{attribute 'ac_persist' := 'PersistenceChannel'}
Low_temperature_alarm_differential : REAL ;
{attribute 'ac_persist' := 'PersistenceChannel'}
High_temperature_alarm_differential : REAL ;
{attribute 'ac_persist' := 'PersistenceChannel'}
Probe_used_for_temperature_alarm_detection : REAL ;
{attribute 'ac_persist' := 'PersistenceChannel'}
Temperature_alarm_delay : REAL ;
Temperature_alarm_delay_write_int : INT ;
{attribute 'ac_persist' := 'PersistenceChannel'}
Operation_in_case_of_high_condenser_alarm : REAL ;
{attribute 'ac_persist' := 'PersistenceChannel'}
Condensation_temperature_alarm : REAL ;
{attribute 'ac_persist' := 'PersistenceChannel'}
Standby_button_enabling : REAL ;
{attribute 'ac_persist' := 'PersistenceChannel'}
Door_switch_input_mode : REAL ;
Door_switch_input_mode_write_int : INT ;
{attribute 'ac_persist' := 'PersistenceChannel'}
Door_alarm_delay : REAL ;
Door_alarm_delay_write_int : INT ;
{attribute 'ac_persist' := 'PersistenceChannel'}
Compressor_stop_delay : REAL ;
Compressor_stop_delay_write_int : INT ;
{attribute 'ac_persist' := 'PersistenceChannel'}
Door_stop_timeout : REAL ;
Door_stop_timeout_write_int : INT ;
{attribute 'ac_persist' := 'PersistenceChannel'}
DI1_digital_input_operation : REAL ;
{attribute 'ac_persist' := 'PersistenceChannel'}
DI1_digital_input_activation : REAL ;
{attribute 'ac_persist' := 'PersistenceChannel'}
DI2_digital_input_operation : REAL ;
{attribute 'ac_persist' := 'PersistenceChannel'}
DI2_digital_input_activation : REAL ;
DI1_digital_input_operation_write_int : INT ;
DI1_digital_input_activation_write_int : INT ;
DI2_digital_input_operation_write_int : INT ;
DI2_digital_input_activation_write_int : INT ;
{attribute 'ac_persist' := 'PersistenceChannel'}
Light_control_mode : REAL ;
Light_control_mode_write_int : INT ;
{attribute 'ac_persist' := 'PersistenceChannel'}
standby : REAL;
standby_write : INT;
{attribute 'ac_persist' := 'PersistenceChannel'}
Light_control : REAL;

write_data_alarm : R_TRIG;
write_data_setp : R_TRIG;
write_data_defrost : R_TRIG;
write_data_mute : R_TRIG;
write_data_control : R_TRIG;
write_data_man_defrost : R_TRIG;
door_open_trigger : R_TRIG ;
door_close_trigger : F_TRIG ;
set_param_trigger : R_TRIG ;
get_param_trigger : R_TRIG ;
all_param_read : BOOL ;
no_loop : INT :=0 ;


control_button : BOOL  := TRUE ;
defrost_button : BOOL  := FALSE ;
setpoint_button : BOOL ;
read_param_button : BOOL ;
{attribute 'ac_persist' := 'PersistenceChannel'}
RL1_output_operation : REAL ;
{attribute 'ac_persist' := 'PersistenceChannel'}
RL2_output_operation : REAL ;
{attribute 'ac_persist' := 'PersistenceChannel'}
RL3_output_operation : REAL ;
{attribute 'ac_persist' := 'PersistenceChannel'}
RL4_output_operation : REAL ;
RL1_output_operation_write_int : INT ;
RL2_output_operation_write_int : INT ;
RL3_output_operation_write_int : INT ;
RL4_output_operation_write_int : INT ;
{attribute 'ac_persist' := 'PersistenceChannel'}
Probe_T1_offset : REAL ;
{attribute 'ac_persist' := 'PersistenceChannel'}
Probe_T2_enable : REAL ;
{attribute 'ac_persist' := 'PersistenceChannel'}
Probe_T2_offset : REAL ;
{attribute 'ac_persist' := 'PersistenceChannel'}
Auxiliary_probe_T3_operation : REAL ;
{attribute 'ac_persist' := 'PersistenceChannel'}
Probe_T3_offset : REAL ;
{attribute 'ac_persist' := 'PersistenceChannel'}
Delay_for_minimum_and_maximum_temperature_logging : REAL ;
{attribute 'ac_persist' := 'PersistenceChannel'}
Selects_the_temperature_probe_to_be_displayed : REAL ;
{attribute 'ac_persist' := 'PersistenceChannel'}
The_relative_weight_of_T2_on_T1 : REAL ;
{attribute 'ac_persist' := 'PersistenceChannel'}
Display_slowdown : REAL ;
Display_slowdown_write_int : INT ;
{attribute 'ac_persist' := 'PersistenceChannel'}
Address_for_PC_communication : REAL ;
Address_for_PC_communication_write_int : INT ;
{attribute 'ac_persist' := 'PersistenceChannel'}
Modbus_protocol_selection : REAL ;
Modbus_protocol_selection_write_int : INT ;
// Word variables
Status_BITs_0_to_15 : WORD;
Status_BITs_16_to_31 : WORD;
Alarm_BITs_0_to_15 : WORD;
setp_write_word : WORD ;
Fan_stop_temperature_write_word : WORD ;

dig1 : BOOL;
dig2 : BOOL;
dout1 : BOOL;
dout2 : BOOL;
dout3 : BOOL;
dout4 : BOOL;
alarm : BOOL;
buzzer_mute : BOOL;
defrost : BOOL;
door_open : BOOL;
test : BOOL;
machine_standby : BOOL;
T1_failure  : BOOL;
T2_failure  : BOOL;
T3_failure  : BOOL;
Low_temperature  : BOOL;
High_temperature  : BOOL;
High_condenser_temperature  : BOOL;
Generic_alarm  : BOOL;
Door_open_alarm  : BOOL;
RL1 : BOOL;
RL2 : BOOL;
RL3 : BOOL;
SSR : BOOL;
deactivate_defrost_button : BOOL ;
modbus_communication : BOOL ;
comm_indicator : REAL ;



//triggers for writing setpoints and parameters
xtrigger_alarm : BOOL;
xtrigger_setp : BOOL;
xtrigger_defrost : BOOL;
xtrigger_mute : BOOL;
xtrigger_control : BOOL;
xtrigger_man_defrost : BOOL;
xtrigger_get_param : BOOL;
xtrigger_set_param : BOOL;







//Graphic variables
Unit_switch_status : INT;
i : INT;
show_trendvalue : ARRAY[0..50] OF BOOL;
select_trendvalue : INT :=0 ;

END_VAR




temp_provision_room:= scaleFunction(modbus_var[0],0.1, 0);
temp_defrost := scaleFunction(modbus_var[1],0.1, 0);
reg2 := scaleFunction(modbus_var[2],0.1, 0); // not used ?
reg3 := scaleFunction(modbus_var[3],0.1, 0); // not used ?
reg4 := scaleFunction(modbus_var[4],0.1, 0); // not used ?
reg5 := scaleFunction(modbus_var[5],0.1, 0); // not used ?
reg6 := scaleFunction(modbus_var[6],0.1, 0); // not used ?
reg7 := scaleFunction(modbus_var[7],0.1, 0); // not used ?
reg8 := scaleFunction(modbus_var[8],0.1, 0); // not used ?
reg9 := scaleFunction(modbus_var[9],0.1, 0); // not used ?
reg10 := modbus_var[10]; // not used ?
set_point := scaleFunction(modbus_var[11],0.1, 0);  // not used ?
reg12 := scaleFunction(modbus_var[12],0.1, 0); // not used ?
reg13 := scaleFunction(modbus_var[13],0.1, 0); // not used ?
reg14 := scaleFunction(modbus_var[14],0.1, 0); // not used ?
reg15 := scaleFunction(modbus_var[15],0.1, 0); // not used ?
reg16 := scaleFunction(modbus_var[16],0.1, 0); // not used ?
reg17 := scaleFunction(modbus_var[17],0.1, 0); // not used ?

// Non changeable parameters

T1_offset := scaleFunction(modbus_var1[2000],1, 0);
T2_offset := scaleFunction(modbus_var1[2001],1, 2);
T3_offset := scaleFunction(modbus_var1[2002],1, 3);
T1_span := scaleFunction(modbus_var1[2003],1, 4);
T2_span := scaleFunction(modbus_var1[2004],1, 5);
T3_span := scaleFunction(modbus_var1[2005],1, 6);

valore_tasto1_V := scaleFunction(modbus_var[150],1, 6);
valore_tasto_UP := scaleFunction(modbus_var[151],1, 6);
valore_tasto_DW := scaleFunction(modbus_var[152],1, 6);
valore_tasto_X := scaleFunction(modbus_var[153],1, 6);

Test_display := scaleFunction(modbus_var[193],1, 0);
Tasto_attualmente_premuto := scaleFunction(modbus_var[194],1, 0);
Password := scaleFunction(modbus_var[197],1, 0);

preset_parameters:= scaleFunction(modbus_var[200],1, 0);

Setpoint:= scaleFunction(modbus_var[303],0.1, 0);
Thermostat_OFF_ON_ref_to_SP:= scaleFunction(modbus_var[304],0.1, 0);
Thermostat_ON_OFF_ref_to_SP:= scaleFunction(modbus_var[305],0.1, 0);

Defrost_start_mode:= scaleFunction(modbus_var[400],1, 0);
Time_based_defrost:= scaleFunction(modbus_var[401],1, 0);

Delay_for_pressure_equalization_for_hot_gas:= scaleFunction(modbus_var[405],1, 0);

Defrost_end_temperature:= scaleFunction(modbus_var[406],0.1, 0);
Maximum_defrost_duration:= scaleFunction(modbus_var[407],1, 0);

Drain_down_time:= scaleFunction(modbus_var[408],1, 0);
Display_defrost_mode:= scaleFunction(modbus_var[409],1, 0);

Target_evaporator_temperature:= scaleFunction(modbus_var[453],0.1, 0);
Fan_stop_delay_after_compressor_stop:= scaleFunction(modbus_var[454],1, 0);
Timed_fan_stop:= scaleFunction(modbus_var[455],1, 0);
Timed_fan_run:= scaleFunction(modbus_var[456],1, 0);
Fan_Minimum_Stop:= scaleFunction(modbus_var[457],1, 0);


Low_temperature_alarm_threshold:= scaleFunction(modbus_var[501],0.1, 0);
High_temperature_alarm_threshold:= scaleFunction(modbus_var[502],0.1, 0);
Low_temperature_alarm_differential:= scaleFunction(modbus_var[503],0.1, 0);
High_temperature_alarm_differential:= scaleFunction(modbus_var[504],0.1, 0);
Probe_used_for_temperature_alarm_detection:= scaleFunction(modbus_var[505],1, 0);
Operation_in_case_of_high_condenser_alarm:= scaleFunction(modbus_var[507],1, 0);
Condensation_temperature_alarm:= scaleFunction(modbus_var[508],0.1, 0);

Standby_button_enabling:= scaleFunction(modbus_var[600],1, 0);



// Changeable parameters
delay_timer(IN:=read_param_button, PT:=set_delaytime);
IF read_param_button THEN
	Display_slowdown:= scaleFunction(modbus_var[208],1, 0);
	Readout_scale:= scaleFunction(modbus_var[300],1, 0);
	Minimum_temperature_setpoint:= scaleFunction(modbus_var[301],0.1, 0);
	Maximum_temperature_setpoint:= scaleFunction(modbus_var[302],0.1, 0);
	CH_minimum_OFF_time:= scaleFunction(modbus_var[306],1, 0);
	CH_minimum_ON_time:= scaleFunction(modbus_var[307],1, 0);
	CH_output_ON_when_probe_T1_is_faulty:= scaleFunction(modbus_var[308],1, 0);
	CH_output_OFF_when_probe_T1_is_faulty:= scaleFunction(modbus_var[309],1, 0);
	Minimum_Time_Between_Defrost:= scaleFunction(modbus_var[402],1, 0);
	Defrost_time_optimization:= scaleFunction(modbus_var[403],1, 0);
	Defrost_type:= scaleFunction(modbus_var[404],1, 0);
//	Defrost_end_temperature:= scaleFunction(modbus_var[406],1, 0);
//	Maximum_defrost_duration:= scaleFunction(modbus_var[407],1, 0);
	Display_delay:= scaleFunction(modbus_var[410],1, 0);
	Fans_active_during_defrost:= scaleFunction(modbus_var[411],1, 0);
	Fan_restart_temperature_after_defrost:= scaleFunction(modbus_var[412],0.1, 0);
	Fan_mode_during_thermostatic_control:= scaleFunction(modbus_var[452],1, 0);
	Fan_stop_temperature:= scaleFunction(modbus_var[450],0.1, 0);
	Maximum_fan_stop_for_FDD_FET:= scaleFunction(modbus_var[451],1, 0);
	Alarm_threshold_management:= scaleFunction(modbus_var[500],1, 0);
	Temperature_alarm_delay:= scaleFunction(modbus_var[506],1, 0);
	Door_switch_input_mode:= scaleFunction(modbus_var[601],1, 0);
	Door_alarm_delay:= scaleFunction(modbus_var[602],1, 0);
	Compressor_stop_delay:= scaleFunction(modbus_var[603],1, 0);
	Door_stop_timeout:= scaleFunction(modbus_var[604],1, 0);
	DI1_digital_input_operation:= scaleFunction(modbus_var[605],1, 0);
	DI1_digital_input_activation:= scaleFunction(modbus_var[606],1, 0);
	DI2_digital_input_operation:= scaleFunction(modbus_var[607],1, 0);
	DI2_digital_input_activation:= scaleFunction(modbus_var[608],1, 0);
	Light_control_mode:= scaleFunction(modbus_var[609],1, 0);
	RL1_output_operation:= scaleFunction(modbus_var[650],1, 0);
	RL2_output_operation:= scaleFunction(modbus_var[651],1, 0);
	RL3_output_operation:= scaleFunction(modbus_var[652],1, 0);
	RL4_output_operation:= scaleFunction(modbus_var[653],1, 0);

	// no_loop :=no_loop +1 ;
	IF delay_timer.Q THEN
		read_param_button := FALSE ;
		no_loop:=0;
	END_IF	
END_IF










standby:= scaleFunction(modbus_var[702],1, 0);
Light_control:= scaleFunction(modbus_var[703],1, 0);




Probe_T1_offset:= scaleFunction(modbus_var[201],0.1, 0);
Probe_T2_enable:= scaleFunction(modbus_var[202],1, 0);
Probe_T2_offset:= scaleFunction(modbus_var[203],0.1, 0);
Auxiliary_probe_T3_operation:= scaleFunction(modbus_var[204],1, 0);
Probe_T3_offset:= scaleFunction(modbus_var[205],0.1, 0);
Selects_the_temperature_probe_to_be_displayed:= scaleFunction(modbus_var[206],1, 0);
The_relative_weight_of_T2_on_T1:= scaleFunction(modbus_var[207],1, 0);

Address_for_PC_communication:= scaleFunction(modbus_var[209],1, 0);
Modbus_protocol_selection:= scaleFunction(modbus_var[210],1, 0);
Delay_for_minimum_and_maximum_temperature_logging:= scaleFunction(modbus_var[211],1, 0);

//  Statusbits
Status_BITs_0_to_15 := modbus_var[100];
Status_BITs_16_to_31 := modbus_var[102];
Alarm_BITs_0_to_15 := modbus_var[101];


alarm := maskbitFunction(Status_BITs_0_to_15,0) OR NOT modbus_communication ;
buzzer_mute := maskbitFunction(Status_BITs_0_to_15,1);
defrost:= maskbitFunction(Status_BITs_0_to_15,2);
door_open := maskbitFunction(Status_BITs_0_to_15,3);
test := maskbitFunction(Status_BITs_0_to_15,4);
machine_standby := maskbitFunction(Status_BITs_0_to_15,5);


T1_failure := maskbitFunction(Alarm_BITs_0_to_15,0);
T2_failure := maskbitFunction(Alarm_BITs_0_to_15,1);
T3_failure := maskbitFunction(Alarm_BITs_0_to_15,2);
Low_temperature := maskbitFunction(Alarm_BITs_0_to_15,3);
High_temperature := maskbitFunction(Alarm_BITs_0_to_15,4);
High_condenser_temperature := maskbitFunction(Alarm_BITs_0_to_15,5);
Generic_alarm := maskbitFunction(Alarm_BITs_0_to_15,6);
Door_open_alarm := maskbitFunction(Alarm_BITs_0_to_15,7);

dout1 := maskbitFunction(Status_BITs_16_to_31,0); 
dout2 := maskbitFunction(Status_BITs_16_to_31,1);
dout3 := maskbitFunction(Status_BITs_16_to_31,2);
dout4 := maskbitFunction(Status_BITs_16_to_31,3);

RL1 := maskbitFunction(modbus_var[196],0);
RL2 := maskbitFunction(modbus_var[196],1);

RL3 := maskbitFunction(modbus_var[196],2);
SSR := maskbitFunction(modbus_var[196],3);


dig1 := maskbitFunction(reg10,0);
dig2 := maskbitFunction(reg10,1);

// Communication fault
comm_indicator := temp_provision_room + temp_defrost + reg2 + reg3 + reg4 + reg5
+ reg6 + reg7 + reg8 + reg9 + reg10 ;
IF comm_indicator = 0 THEN
	modbus_communication := FALSE ;
ELSE
	modbus_communication := TRUE ;
END_IF
	



// Parameter write values

setp_write_word := REAL_TO_INT(setp_write*10) ;
Thermostat_OFF_ON_write_word := REAL_TO_INT(Thermostat_OFF_ON_write*10) ;
Thermostat_ON_OFF_write_word:= REAL_TO_INT(Thermostat_ON_OFF_write*10) ;
Low_temperature_alarm_thres_write_word:= REAL_TO_INT(Low_temperature_alarm_thres_write*10);
High_temperature_alarm_thres_write_word:= REAL_TO_INT(High_temperature_alarm_thres_write*10);
muteAlarm :=1 ;
Time_based_defrost_write_word:= REAL_TO_INT(Time_based_defrost_write*1);
Defrost_end_temperature_write_word:= REAL_TO_INT(Defrost_end_temperature_write*10);
Drain_down_time_write_int:= REAL_TO_INT(Drain_down_time_write);
Maximum_defrost_duration_write_word:= REAL_TO_INT(Maximum_defrost_duration_write*1);
Fan_stop_temperature_write_word:= REAL_TO_INT(Fan_stop_temperature*10);
preset_parameters_write_int:=REAL_TO_INT(preset_parameters);
Readout_scale_write_int:=REAL_TO_INT(Readout_scale);
Minimum_temperature_setpoint_write_int:=REAL_TO_INT(Minimum_temperature_setpoint*10);
Maximum_temperature_setpoint_write_int:=REAL_TO_INT(Maximum_temperature_setpoint*10);
CH_minimum_OFF_time_write_int:=REAL_TO_INT(CH_minimum_OFF_time);
CH_minimum_ON_time_write_int:=REAL_TO_INT(CH_minimum_ON_time);
CH_output_ON_when_probe_T1_is_faulty_write_int:=REAL_TO_INT(CH_output_ON_when_probe_T1_is_faulty);
CH_output_OFF_when_probe_T1_is_faulty_write_int:=REAL_TO_INT(CH_output_OFF_when_probe_T1_is_faulty);
Minimum_Time_Between_Defrost_write_int:=REAL_TO_INT(Minimum_Time_Between_Defrost);
Defrost_time_optimization_write_int:=REAL_TO_INT(Defrost_time_optimization);
Defrost_type_write_int:=REAL_TO_INT(Defrost_type);
Display_delay_write_int:=REAL_TO_INT(Display_delay);
Fans_active_during_defrost_write_int:=REAL_TO_INT(Fans_active_during_defrost);
Fan_restart_temperature_after_defrost_write_int:=REAL_TO_INT(Fan_restart_temperature_after_defrost*10);
// Fan_stop_temperature_write_int:=REAL_TO_INT(Fan_stop_temperature);
Maximum_fan_stop_for_FDD_FET_write_int:=REAL_TO_INT(Maximum_fan_stop_for_FDD_FET);
Fan_mode_during_thermostatic_control_write_int:=REAL_TO_INT(Fan_mode_during_thermostatic_control);
Alarm_threshold_management_write_int:=REAL_TO_INT(Alarm_threshold_management);
Temperature_alarm_delay_write_int:=REAL_TO_INT(Temperature_alarm_delay);
Door_switch_input_mode_write_int:=REAL_TO_INT(Door_switch_input_mode);
Door_alarm_delay_write_int:=REAL_TO_INT(Door_alarm_delay);
Compressor_stop_delay_write_int:=REAL_TO_INT(Compressor_stop_delay);
Door_stop_timeout_write_int:=REAL_TO_INT(Door_stop_timeout);
DI1_digital_input_operation_write_int:=REAL_TO_INT(DI1_digital_input_operation);
DI1_digital_input_activation_write_int:=REAL_TO_INT(DI1_digital_input_activation);
DI2_digital_input_operation_write_int:=REAL_TO_INT(DI2_digital_input_operation);
DI2_digital_input_activation_write_int:=REAL_TO_INT(DI2_digital_input_activation);
Light_control_mode_write_int:=REAL_TO_INT(Light_control_mode);
RL1_output_operation_write_int:=REAL_TO_INT(RL1_output_operation);
RL2_output_operation_write_int:=REAL_TO_INT(RL2_output_operation);
RL3_output_operation_write_int:=REAL_TO_INT(RL3_output_operation);
RL4_output_operation_write_int:=REAL_TO_INT(RL4_output_operation);
Display_slowdown_write_int:=REAL_TO_INT(Display_slowdown);
Address_for_PC_communication_write_int:=REAL_TO_INT(Address_for_PC_communication);
Modbus_protocol_selection_write_int:=REAL_TO_INT(Modbus_protocol_selection);

write_data_alarm(clk:=xtrigger_alarm);
write_data_setp(clk:=xtrigger_setp);
write_data_defrost(clk:=xtrigger_defrost);
write_data_mute(clk:=xtrigger_mute);
write_data_control(clk:=xtrigger_control);
write_data_man_defrost(clk:=xtrigger_man_defrost);
get_param_trigger(clk:=xtrigger_get_param);
set_param_trigger(clk:=xtrigger_set_param);


IF control_button THEN
	standby_write := 0 ;
	IF machine_standby=TRUE THEN
		xtrigger_control := TRUE;
	END_IF
ELSE
	standby_write := 1 ;
	IF machine_standby=FALSE THEN
		xtrigger_control := TRUE;
	END_IF	
END_IF


IF defrost_button THEN
	defrost_write := 1 ;
	IF defrost=FALSE THEN
		xtrigger_man_defrost := TRUE;
	END_IF
ELSE
	defrost_write := 0 ;

END_IF

// Door open timers
door_open_trigger(clk:=door_open);
door_close_trigger(clk:=door_open);

timer_door_open(IN:=timer_enable, PT:=T#30D);
timer_door_closed(IN:=timer2_enable, PT:=T#30D);

IF door_open_trigger.Q THEN
	closetime_tot := opentime_tot + timer_door_closed.ET;
	timer_enable := TRUE;
	timer2_enable := FALSE;
END_IF

IF door_close_trigger.Q THEN
	opentime_tot := opentime_tot + timer_door_open.ET;
	timer_enable := FALSE;
	timer2_enable := TRUE ;
END_IF


total_time := opentime_tot + closetime_tot ;

opentime_ms := TO_LREAL(TO_UDINT(opentime_tot) / 1000.0);
totaltime_ms := TO_LREAL(TO_UDINT(total_time) / 1000.0);

opentime_proc := (opentime_ms /totaltime_ms)*100 ;
IF resettimer_button THEN
	opentime_tot := T#0S ;
	closetime_tot := T#0S ;
	total_time := T#0S;
END_IF






// Graphic controls
IF select_trendvalue > 0 THEN
	show_trendvalue[select_trendvalue]:= TRUE;
ELSIF select_trendvalue = 0 THEN
	FOR i := 0 TO 50 DO
      show_trendvalue[i] := FALSE;
   	END_FOR
END_IF ;

END_PROGRAM

// Device/Application/Provision_3
PROGRAM Provision_3
VAR



modbus_var : ARRAY[0..800] OF WORD;
modbus_var1 : ARRAY[2000..2010] OF WORD;
timer_door_open : TON ;
timer_door_closed : TON ;
delay_timer : TON ;
open_time : TIME ;
total_time : TIME ;
opentime_tot : TIME ;
opentime_proc : REAL ;
closetime_tot : TIME ; 
{attribute 'ac_persist' := 'PersistenceChannel'}
set_delaytime : TIME := T#1S;
timer_enable : BOOL;
timer2_enable : BOOL;
timer_elapsed : BOOL ;
start_timer : BOOL := TRUE;
doorclose : F_TRIG;
resettimer_button :BOOL ;
totaltime_ms : LREAL ;
opentime_ms : LREAL ;

temp_provision_room : REAL;
temp_defrost : REAL;
regulator_temp : REAL;

set_point: REAL;
reg2 : REAL ;
reg3 : REAL ;
reg4 : REAL ;
reg5 : REAL ;
reg6 : REAL ;
reg7 : REAL ;
reg8 : REAL ;
reg9 : REAL ;
reg10 : WORD ;
reg11 : REAL ;
reg12 : REAL ;
reg13 : REAL ;
reg14 : REAL ;
reg15 : REAL ;
reg16 : REAL ;
reg17 : REAL ;
T1_offset : REAL ;
T2_offset : REAL ;
T3_offset : REAL ;
T1_span : REAL ;
T2_span : REAL ;
T3_span : REAL ;
valore_tasto1_V : REAL ;
valore_tasto_UP : REAL ;
valore_tasto_DW : REAL ;
valore_tasto_X : REAL ;
Test_display : REAL ;
Tasto_attualmente_premuto : REAL ;
Password : REAL ;

{attribute 'ac_persist' := 'PersistenceChannel'}
preset_parameters : REAL ;
preset_parameters_write_int :INT;
{attribute 'ac_persist' := 'PersistenceChannel'}
Readout_scale : REAL ;
{attribute 'ac_persist' := 'PersistenceChannel'}
Readout_scale_write_int : INT;
{attribute 'ac_persist' := 'PersistenceChannel'}
Minimum_temperature_setpoint : REAL ;
Minimum_temperature_setpoint_write_int : INT ;
{attribute 'ac_persist' := 'PersistenceChannel'}
Maximum_temperature_setpoint : REAL ;
Maximum_temperature_setpoint_write_int : INT ;
setp_write : REAL ;
{attribute 'ac_persist' := 'PersistenceChannel'}
Setpoint : REAL ;
{attribute 'ac_persist' := 'PersistenceChannel'}
Thermostat_OFF_ON_ref_to_SP : REAL  ;
{attribute 'ac_persist' := 'PersistenceChannel'}
Thermostat_ON_OFF_ref_to_SP : REAL  ;
Thermostat_OFF_ON_write : REAL  := 1.0 ;
Thermostat_ON_OFF_write : REAL  := 1.0 ;
Thermostat_OFF_ON_write_word : WORD ;
Thermostat_ON_OFF_write_word : WORD ;
Time_based_defrost_write : REAL   := 8.0  ;
Time_based_defrost_write_word : WORD  ;
Defrost_end_temperature_write : REAL  := 20.0 ;
Defrost_end_temperature_write_word : WORD ;
Fan_restart_temperature_after_defrost_write : REAL ;
Fan_restart_temperature_after_defrost_write_int : INT ;
Maximum_defrost_duration_write : REAL ;
Maximum_defrost_duration_write_word : WORD ;
defrost_write : WORD :=0 ;
{attribute 'ac_persist' := 'PersistenceChannel'}
CH_minimum_OFF_time : REAL ;
CH_minimum_OFF_time_write_int : INT ;
{attribute 'ac_persist' := 'PersistenceChannel'}
CH_minimum_ON_time : REAL ;
CH_minimum_ON_time_write_int : INT ;
{attribute 'ac_persist' := 'PersistenceChannel'}
CH_output_ON_when_probe_T1_is_faulty : REAL ;
CH_output_ON_when_probe_T1_is_faulty_write_int : INT ;
{attribute 'ac_persist' := 'PersistenceChannel'}
CH_output_OFF_when_probe_T1_is_faulty : REAL ;
CH_output_OFF_when_probe_T1_is_faulty_write_int : INT ;

{attribute 'ac_persist' := 'PersistenceChannel'}
Defrost_start_mode : REAL ;
{attribute 'ac_persist' := 'PersistenceChannel'}
Time_based_defrost : REAL ;
{attribute 'ac_persist' := 'PersistenceChannel'}
Minimum_Time_Between_Defrost : REAL ;
Minimum_Time_Between_Defrost_write_int : INT;
{attribute 'ac_persist' := 'PersistenceChannel'}
Defrost_time_optimization : REAL ;
Defrost_time_optimization_write_int : INT;
{attribute 'ac_persist' := 'PersistenceChannel'}
Defrost_type : REAL ;
Defrost_type_write_int : INT;
{attribute 'ac_persist' := 'PersistenceChannel'}
Delay_for_pressure_equalization_for_hot_gas : REAL ;
{attribute 'ac_persist' := 'PersistenceChannel'}
Defrost_end_temperature : REAL ;
{attribute 'ac_persist' := 'PersistenceChannel'}
Maximum_defrost_duration : REAL ;
{attribute 'ac_persist' := 'PersistenceChannel'}
Drain_down_time : REAL ;
Drain_down_time_write : REAL;
Drain_down_time_write_int : INT;
{attribute 'ac_persist' := 'PersistenceChannel'}
Display_defrost_mode : REAL ;
{attribute 'ac_persist' := 'PersistenceChannel'}
Display_delay : REAL ;
Display_delay_write_int : INT;
{attribute 'ac_persist' := 'PersistenceChannel'}
Fans_active_during_defrost : REAL ;
Fans_active_during_defrost_write_int : INT;
{attribute 'ac_persist' := 'PersistenceChannel'}
Fan_restart_temperature_after_defrost : REAL ;
{attribute 'ac_persist' := 'PersistenceChannel'}
Fan_stop_temperature : REAL ;
Fan_stop_temperature_write_int : INT ;
{attribute 'ac_persist' := 'PersistenceChannel'}
Maximum_fan_stop_for_FDD_FET : REAL ;
Maximum_fan_stop_for_FDD_FET_write_int : INT ;
{attribute 'ac_persist' := 'PersistenceChannel'}
Fan_mode_during_thermostatic_control : REAL ;
Fan_mode_during_thermostatic_control_write_int : INT ;
{attribute 'ac_persist' := 'PersistenceChannel'}
Target_evaporator_temperature : REAL ;
{attribute 'ac_persist' := 'PersistenceChannel'}
Fan_stop_delay_after_compressor_stop : REAL ;
{attribute 'ac_persist' := 'PersistenceChannel'}
Timed_fan_stop : REAL ;
{attribute 'ac_persist' := 'PersistenceChannel'}
Timed_fan_run : REAL ;
{attribute 'ac_persist' := 'PersistenceChannel'}
Fan_Minimum_Stop : REAL ;
{attribute 'ac_persist' := 'PersistenceChannel'}
Alarm_threshold_management : REAL ;
Alarm_threshold_management_write_int : INT ;
{attribute 'ac_persist' := 'PersistenceChannel'}
Low_temperature_alarm_threshold : REAL ;
{attribute 'ac_persist' := 'PersistenceChannel'}
High_temperature_alarm_threshold : REAL ;
Low_temperature_alarm_thres_write  : REAL := -20.0 ;
High_temperature_alarm_thres_write : REAL := 20.0 ;
Low_temperature_alarm_thres_write_word : WORD ;
High_temperature_alarm_thres_write_word : WORD ;
muteAlarm : WORD := 1;

{attribute 'ac_persist' := 'PersistenceChannel'}
Low_temperature_alarm_differential : REAL ;
{attribute 'ac_persist' := 'PersistenceChannel'}
High_temperature_alarm_differential : REAL ;
{attribute 'ac_persist' := 'PersistenceChannel'}
Probe_used_for_temperature_alarm_detection : REAL ;
{attribute 'ac_persist' := 'PersistenceChannel'}
Temperature_alarm_delay : REAL ;
Temperature_alarm_delay_write_int : INT ;
{attribute 'ac_persist' := 'PersistenceChannel'}
Operation_in_case_of_high_condenser_alarm : REAL ;
{attribute 'ac_persist' := 'PersistenceChannel'}
Condensation_temperature_alarm : REAL ;
{attribute 'ac_persist' := 'PersistenceChannel'}
Standby_button_enabling : REAL ;
{attribute 'ac_persist' := 'PersistenceChannel'}
Door_switch_input_mode : REAL ;
Door_switch_input_mode_write_int : INT ;
{attribute 'ac_persist' := 'PersistenceChannel'}
Door_alarm_delay : REAL ;
Door_alarm_delay_write_int : INT ;
{attribute 'ac_persist' := 'PersistenceChannel'}
Compressor_stop_delay : REAL ;
Compressor_stop_delay_write_int : INT ;
{attribute 'ac_persist' := 'PersistenceChannel'}
Door_stop_timeout : REAL ;
Door_stop_timeout_write_int : INT ;
{attribute 'ac_persist' := 'PersistenceChannel'}
DI1_digital_input_operation : REAL ;
{attribute 'ac_persist' := 'PersistenceChannel'}
DI1_digital_input_activation : REAL ;
{attribute 'ac_persist' := 'PersistenceChannel'}
DI2_digital_input_operation : REAL ;
{attribute 'ac_persist' := 'PersistenceChannel'}
DI2_digital_input_activation : REAL ;
DI1_digital_input_operation_write_int : INT ;
DI1_digital_input_activation_write_int : INT ;
DI2_digital_input_operation_write_int : INT ;
DI2_digital_input_activation_write_int : INT ;
{attribute 'ac_persist' := 'PersistenceChannel'}
Light_control_mode : REAL ;
Light_control_mode_write_int : INT ;
{attribute 'ac_persist' := 'PersistenceChannel'}
standby : REAL;
standby_write : INT;
{attribute 'ac_persist' := 'PersistenceChannel'}
Light_control : REAL;

write_data_alarm : R_TRIG;
write_data_setp : R_TRIG;
write_data_defrost : R_TRIG;
write_data_mute : R_TRIG;
write_data_control : R_TRIG;
write_data_man_defrost : R_TRIG;
door_open_trigger : R_TRIG ;
door_close_trigger : F_TRIG ;
set_param_trigger : R_TRIG ;
get_param_trigger : R_TRIG ;
all_param_read : BOOL ;
no_loop : INT :=0 ;


control_button : BOOL  := TRUE ;
defrost_button : BOOL  := FALSE ;
setpoint_button : BOOL ;
read_param_button : BOOL ;
{attribute 'ac_persist' := 'PersistenceChannel'}
RL1_output_operation : REAL ;
{attribute 'ac_persist' := 'PersistenceChannel'}
RL2_output_operation : REAL ;
{attribute 'ac_persist' := 'PersistenceChannel'}
RL3_output_operation : REAL ;
{attribute 'ac_persist' := 'PersistenceChannel'}
RL4_output_operation : REAL ;
RL1_output_operation_write_int : INT ;
RL2_output_operation_write_int : INT ;
RL3_output_operation_write_int : INT ;
RL4_output_operation_write_int : INT ;
{attribute 'ac_persist' := 'PersistenceChannel'}
Probe_T1_offset : REAL ;
{attribute 'ac_persist' := 'PersistenceChannel'}
Probe_T2_enable : REAL ;
{attribute 'ac_persist' := 'PersistenceChannel'}
Probe_T2_offset : REAL ;
{attribute 'ac_persist' := 'PersistenceChannel'}
Auxiliary_probe_T3_operation : REAL ;
{attribute 'ac_persist' := 'PersistenceChannel'}
Probe_T3_offset : REAL ;
{attribute 'ac_persist' := 'PersistenceChannel'}
Delay_for_minimum_and_maximum_temperature_logging : REAL ;
{attribute 'ac_persist' := 'PersistenceChannel'}
Selects_the_temperature_probe_to_be_displayed : REAL ;
{attribute 'ac_persist' := 'PersistenceChannel'}
The_relative_weight_of_T2_on_T1 : REAL ;
{attribute 'ac_persist' := 'PersistenceChannel'}
Display_slowdown : REAL ;
Display_slowdown_write_int : INT ;
{attribute 'ac_persist' := 'PersistenceChannel'}
Address_for_PC_communication : REAL ;
Address_for_PC_communication_write_int : INT ;
{attribute 'ac_persist' := 'PersistenceChannel'}
Modbus_protocol_selection : REAL ;
Modbus_protocol_selection_write_int : INT ;
// Word variables
Status_BITs_0_to_15 : WORD;
Status_BITs_16_to_31 : WORD;
Alarm_BITs_0_to_15 : WORD;
setp_write_word : WORD ;
Fan_stop_temperature_write_word : WORD ;

dig1 : BOOL;
dig2 : BOOL;
dout1 : BOOL;
dout2 : BOOL;
dout3 : BOOL;
dout4 : BOOL;
alarm : BOOL;
buzzer_mute : BOOL;
defrost : BOOL;
door_open : BOOL;
test : BOOL;
machine_standby : BOOL;
T1_failure  : BOOL;
T2_failure  : BOOL;
T3_failure  : BOOL;
Low_temperature  : BOOL;
High_temperature  : BOOL;
High_condenser_temperature  : BOOL;
Generic_alarm  : BOOL;
Door_open_alarm  : BOOL;
RL1 : BOOL;
RL2 : BOOL;
RL3 : BOOL;
SSR : BOOL;
deactivate_defrost_button : BOOL ;
modbus_communication : BOOL ;
comm_indicator : REAL ;



//triggers for writing setpoints and parameters
xtrigger_alarm : BOOL;
xtrigger_setp : BOOL;
xtrigger_defrost : BOOL;
xtrigger_mute : BOOL;
xtrigger_control : BOOL;
xtrigger_man_defrost : BOOL;
xtrigger_get_param : BOOL;
xtrigger_set_param : BOOL;








//Graphic variables
Unit_switch_status : INT;
i : INT;
show_trendvalue : ARRAY[0..50] OF BOOL;
select_trendvalue : INT :=0 ;

END_VAR




temp_provision_room:= scaleFunction(modbus_var[0],0.1, 0);
temp_defrost := scaleFunction(modbus_var[1],0.1, 0);
reg2 := scaleFunction(modbus_var[2],0.1, 0); // not used ?
reg3 := scaleFunction(modbus_var[3],0.1, 0); // not used ?
reg4 := scaleFunction(modbus_var[4],0.1, 0); // not used ?
reg5 := scaleFunction(modbus_var[5],0.1, 0); // not used ?
reg6 := scaleFunction(modbus_var[6],0.1, 0); // not used ?
reg7 := scaleFunction(modbus_var[7],0.1, 0); // not used ?
reg8 := scaleFunction(modbus_var[8],0.1, 0); // not used ?
reg9 := scaleFunction(modbus_var[9],0.1, 0); // not used ?
reg10 := modbus_var[10]; // not used ?
set_point := scaleFunction(modbus_var[11],0.1, 0);  // not used ?
reg12 := scaleFunction(modbus_var[12],0.1, 0); // not used ?
reg13 := scaleFunction(modbus_var[13],0.1, 0); // not used ?
reg14 := scaleFunction(modbus_var[14],0.1, 0); // not used ?
reg15 := scaleFunction(modbus_var[15],0.1, 0); // not used ?
reg16 := scaleFunction(modbus_var[16],0.1, 0); // not used ?
reg17 := scaleFunction(modbus_var[17],0.1, 0); // not used ?

// Non changeable parameters

T1_offset := scaleFunction(modbus_var1[2000],1, 0);
T2_offset := scaleFunction(modbus_var1[2001],1, 2);
T3_offset := scaleFunction(modbus_var1[2002],1, 3);
T1_span := scaleFunction(modbus_var1[2003],1, 4);
T2_span := scaleFunction(modbus_var1[2004],1, 5);
T3_span := scaleFunction(modbus_var1[2005],1, 6);

valore_tasto1_V := scaleFunction(modbus_var[150],1, 6);
valore_tasto_UP := scaleFunction(modbus_var[151],1, 6);
valore_tasto_DW := scaleFunction(modbus_var[152],1, 6);
valore_tasto_X := scaleFunction(modbus_var[153],1, 6);

Test_display := scaleFunction(modbus_var[193],1, 0);
Tasto_attualmente_premuto := scaleFunction(modbus_var[194],1, 0);
Password := scaleFunction(modbus_var[197],1, 0);

preset_parameters:= scaleFunction(modbus_var[200],1, 0);

Setpoint:= scaleFunction(modbus_var[303],0.1, 0);
Thermostat_OFF_ON_ref_to_SP:= scaleFunction(modbus_var[304],0.1, 0);
Thermostat_ON_OFF_ref_to_SP:= scaleFunction(modbus_var[305],0.1, 0);

Defrost_start_mode:= scaleFunction(modbus_var[400],1, 0);
Time_based_defrost:= scaleFunction(modbus_var[401],1, 0);

Delay_for_pressure_equalization_for_hot_gas:= scaleFunction(modbus_var[405],1, 0);

Defrost_end_temperature:= scaleFunction(modbus_var[406],0.1, 0);
Maximum_defrost_duration:= scaleFunction(modbus_var[407],1, 0);

Drain_down_time:= scaleFunction(modbus_var[408],1, 0);
Display_defrost_mode:= scaleFunction(modbus_var[409],1, 0);

Target_evaporator_temperature:= scaleFunction(modbus_var[453],0.1, 0);
Fan_stop_delay_after_compressor_stop:= scaleFunction(modbus_var[454],1, 0);
Timed_fan_stop:= scaleFunction(modbus_var[455],1, 0);
Timed_fan_run:= scaleFunction(modbus_var[456],1, 0);
Fan_Minimum_Stop:= scaleFunction(modbus_var[457],1, 0);


Low_temperature_alarm_threshold:= scaleFunction(modbus_var[501],0.1, 0);
High_temperature_alarm_threshold:= scaleFunction(modbus_var[502],0.1, 0);
Low_temperature_alarm_differential:= scaleFunction(modbus_var[503],0.1, 0);
High_temperature_alarm_differential:= scaleFunction(modbus_var[504],0.1, 0);
Probe_used_for_temperature_alarm_detection:= scaleFunction(modbus_var[505],1, 0);
Operation_in_case_of_high_condenser_alarm:= scaleFunction(modbus_var[507],1, 0);
Condensation_temperature_alarm:= scaleFunction(modbus_var[508],0.1, 0);

Standby_button_enabling:= scaleFunction(modbus_var[600],1, 0);



// Changeable parameters
delay_timer(IN:=read_param_button, PT:=set_delaytime);
IF read_param_button THEN
	Display_slowdown:= scaleFunction(modbus_var[208],1, 0);
	Readout_scale:= scaleFunction(modbus_var[300],1, 0);
	Minimum_temperature_setpoint:= scaleFunction(modbus_var[301],0.1, 0);
	Maximum_temperature_setpoint:= scaleFunction(modbus_var[302],0.1, 0);
	CH_minimum_OFF_time:= scaleFunction(modbus_var[306],1, 0);
	CH_minimum_ON_time:= scaleFunction(modbus_var[307],1, 0);
	CH_output_ON_when_probe_T1_is_faulty:= scaleFunction(modbus_var[308],1, 0);
	CH_output_OFF_when_probe_T1_is_faulty:= scaleFunction(modbus_var[309],1, 0);
	Minimum_Time_Between_Defrost:= scaleFunction(modbus_var[402],1, 0);
	Defrost_time_optimization:= scaleFunction(modbus_var[403],1, 0);
	Defrost_type:= scaleFunction(modbus_var[404],1, 0);
//	Defrost_end_temperature:= scaleFunction(modbus_var[406],1, 0);
//	Maximum_defrost_duration:= scaleFunction(modbus_var[407],1, 0);
	Display_delay:= scaleFunction(modbus_var[410],1, 0);
	Fans_active_during_defrost:= scaleFunction(modbus_var[411],1, 0);
	Fan_restart_temperature_after_defrost:= scaleFunction(modbus_var[412],0.1, 0);
	Fan_mode_during_thermostatic_control:= scaleFunction(modbus_var[452],1, 0);
	Fan_stop_temperature:= scaleFunction(modbus_var[450],0.1, 0);
	Maximum_fan_stop_for_FDD_FET:= scaleFunction(modbus_var[451],1, 0);
	Alarm_threshold_management:= scaleFunction(modbus_var[500],1, 0);
	Temperature_alarm_delay:= scaleFunction(modbus_var[506],1, 0);
	Door_switch_input_mode:= scaleFunction(modbus_var[601],1, 0);
	Door_alarm_delay:= scaleFunction(modbus_var[602],1, 0);
	Compressor_stop_delay:= scaleFunction(modbus_var[603],1, 0);
	Door_stop_timeout:= scaleFunction(modbus_var[604],1, 0);
	DI1_digital_input_operation:= scaleFunction(modbus_var[605],1, 0);
	DI1_digital_input_activation:= scaleFunction(modbus_var[606],1, 0);
	DI2_digital_input_operation:= scaleFunction(modbus_var[607],1, 0);
	DI2_digital_input_activation:= scaleFunction(modbus_var[608],1, 0);
	Light_control_mode:= scaleFunction(modbus_var[609],1, 0);
	RL1_output_operation:= scaleFunction(modbus_var[650],1, 0);
	RL2_output_operation:= scaleFunction(modbus_var[651],1, 0);
	RL3_output_operation:= scaleFunction(modbus_var[652],1, 0);
	RL4_output_operation:= scaleFunction(modbus_var[653],1, 0);

	// no_loop :=no_loop +1 ;
	IF delay_timer.Q THEN
		read_param_button := FALSE ;
		no_loop:=0;
	END_IF	
END_IF










standby:= scaleFunction(modbus_var[702],1, 0);
Light_control:= scaleFunction(modbus_var[703],1, 0);




Probe_T1_offset:= scaleFunction(modbus_var[201],0.1, 0);
Probe_T2_enable:= scaleFunction(modbus_var[202],1, 0);
Probe_T2_offset:= scaleFunction(modbus_var[203],0.1, 0);
Auxiliary_probe_T3_operation:= scaleFunction(modbus_var[204],1, 0);
Probe_T3_offset:= scaleFunction(modbus_var[205],0.1, 0);
Selects_the_temperature_probe_to_be_displayed:= scaleFunction(modbus_var[206],1, 0);
The_relative_weight_of_T2_on_T1:= scaleFunction(modbus_var[207],1, 0);

Address_for_PC_communication:= scaleFunction(modbus_var[209],1, 0);
Modbus_protocol_selection:= scaleFunction(modbus_var[210],1, 0);
Delay_for_minimum_and_maximum_temperature_logging:= scaleFunction(modbus_var[211],1, 0);

//  Statusbits
Status_BITs_0_to_15 := modbus_var[100];
Status_BITs_16_to_31 := modbus_var[102];
Alarm_BITs_0_to_15 := modbus_var[101];


alarm := maskbitFunction(Status_BITs_0_to_15,0) OR NOT modbus_communication ;
buzzer_mute := maskbitFunction(Status_BITs_0_to_15,1);
defrost:= maskbitFunction(Status_BITs_0_to_15,2);
door_open := maskbitFunction(Status_BITs_0_to_15,3);
test := maskbitFunction(Status_BITs_0_to_15,4);
machine_standby := maskbitFunction(Status_BITs_0_to_15,5);


T1_failure := maskbitFunction(Alarm_BITs_0_to_15,0);
T2_failure := maskbitFunction(Alarm_BITs_0_to_15,1);
T3_failure := maskbitFunction(Alarm_BITs_0_to_15,2);
Low_temperature := maskbitFunction(Alarm_BITs_0_to_15,3);
High_temperature := maskbitFunction(Alarm_BITs_0_to_15,4);
High_condenser_temperature := maskbitFunction(Alarm_BITs_0_to_15,5);
Generic_alarm := maskbitFunction(Alarm_BITs_0_to_15,6);
Door_open_alarm := maskbitFunction(Alarm_BITs_0_to_15,7);

dout1 := maskbitFunction(Status_BITs_16_to_31,0); 
dout2 := maskbitFunction(Status_BITs_16_to_31,1);
dout3 := maskbitFunction(Status_BITs_16_to_31,2);
dout4 := maskbitFunction(Status_BITs_16_to_31,3);

RL1 := maskbitFunction(modbus_var[196],0);
RL2 := maskbitFunction(modbus_var[196],1);

RL3 := maskbitFunction(modbus_var[196],2);
SSR := maskbitFunction(modbus_var[196],3);


dig1 := maskbitFunction(reg10,0);
dig2 := maskbitFunction(reg10,1);

// Communication fault
comm_indicator := temp_provision_room + temp_defrost + reg2 + reg3 + reg4 + reg5
+ reg6 + reg7 + reg8 + reg9 + reg10 ;
IF comm_indicator = 0 THEN
	modbus_communication := FALSE ;
ELSE
	modbus_communication := TRUE ;
END_IF
	



// Parameter write values

setp_write_word := REAL_TO_INT(setp_write*10) ;
Thermostat_OFF_ON_write_word := REAL_TO_INT(Thermostat_OFF_ON_write*10) ;
Thermostat_ON_OFF_write_word:= REAL_TO_INT(Thermostat_ON_OFF_write*10) ;
Low_temperature_alarm_thres_write_word:= REAL_TO_INT(Low_temperature_alarm_thres_write*10);
High_temperature_alarm_thres_write_word:= REAL_TO_INT(High_temperature_alarm_thres_write*10);
muteAlarm :=1 ;
Time_based_defrost_write_word:= REAL_TO_INT(Time_based_defrost_write*1);
Defrost_end_temperature_write_word:= REAL_TO_INT(Defrost_end_temperature_write*10);
Drain_down_time_write_int:= REAL_TO_INT(Drain_down_time_write);
Maximum_defrost_duration_write_word:= REAL_TO_INT(Maximum_defrost_duration_write*1);
Fan_stop_temperature_write_word:= REAL_TO_INT(Fan_stop_temperature*10);
preset_parameters_write_int:=REAL_TO_INT(preset_parameters);
Readout_scale_write_int:=REAL_TO_INT(Readout_scale);
Minimum_temperature_setpoint_write_int:=REAL_TO_INT(Minimum_temperature_setpoint*10);
Maximum_temperature_setpoint_write_int:=REAL_TO_INT(Maximum_temperature_setpoint*10);
CH_minimum_OFF_time_write_int:=REAL_TO_INT(CH_minimum_OFF_time);
CH_minimum_ON_time_write_int:=REAL_TO_INT(CH_minimum_ON_time);
CH_output_ON_when_probe_T1_is_faulty_write_int:=REAL_TO_INT(CH_output_ON_when_probe_T1_is_faulty);
CH_output_OFF_when_probe_T1_is_faulty_write_int:=REAL_TO_INT(CH_output_OFF_when_probe_T1_is_faulty);
Minimum_Time_Between_Defrost_write_int:=REAL_TO_INT(Minimum_Time_Between_Defrost);
Defrost_time_optimization_write_int:=REAL_TO_INT(Defrost_time_optimization);
Defrost_type_write_int:=REAL_TO_INT(Defrost_type);
Display_delay_write_int:=REAL_TO_INT(Display_delay);
Fans_active_during_defrost_write_int:=REAL_TO_INT(Fans_active_during_defrost);
Fan_restart_temperature_after_defrost_write_int:=REAL_TO_INT(Fan_restart_temperature_after_defrost*10);
// Fan_stop_temperature_write_int:=REAL_TO_INT(Fan_stop_temperature);
Maximum_fan_stop_for_FDD_FET_write_int:=REAL_TO_INT(Maximum_fan_stop_for_FDD_FET);
Fan_mode_during_thermostatic_control_write_int:=REAL_TO_INT(Fan_mode_during_thermostatic_control);
Alarm_threshold_management_write_int:=REAL_TO_INT(Alarm_threshold_management);
Temperature_alarm_delay_write_int:=REAL_TO_INT(Temperature_alarm_delay);
Door_switch_input_mode_write_int:=REAL_TO_INT(Door_switch_input_mode);
Door_alarm_delay_write_int:=REAL_TO_INT(Door_alarm_delay);
Compressor_stop_delay_write_int:=REAL_TO_INT(Compressor_stop_delay);
Door_stop_timeout_write_int:=REAL_TO_INT(Door_stop_timeout);
DI1_digital_input_operation_write_int:=REAL_TO_INT(DI1_digital_input_operation);
DI1_digital_input_activation_write_int:=REAL_TO_INT(DI1_digital_input_activation);
DI2_digital_input_operation_write_int:=REAL_TO_INT(DI2_digital_input_operation);
DI2_digital_input_activation_write_int:=REAL_TO_INT(DI2_digital_input_activation);
Light_control_mode_write_int:=REAL_TO_INT(Light_control_mode);
RL1_output_operation_write_int:=REAL_TO_INT(RL1_output_operation);
RL2_output_operation_write_int:=REAL_TO_INT(RL2_output_operation);
RL3_output_operation_write_int:=REAL_TO_INT(RL3_output_operation);
RL4_output_operation_write_int:=REAL_TO_INT(RL4_output_operation);
Display_slowdown_write_int:=REAL_TO_INT(Display_slowdown);
Address_for_PC_communication_write_int:=REAL_TO_INT(Address_for_PC_communication);
Modbus_protocol_selection_write_int:=REAL_TO_INT(Modbus_protocol_selection);

write_data_alarm(clk:=xtrigger_alarm);
write_data_setp(clk:=xtrigger_setp);
write_data_defrost(clk:=xtrigger_defrost);
write_data_mute(clk:=xtrigger_mute);
write_data_control(clk:=xtrigger_control);
write_data_man_defrost(clk:=xtrigger_man_defrost);
get_param_trigger(clk:=xtrigger_get_param);
set_param_trigger(clk:=xtrigger_set_param);


IF control_button THEN
	standby_write := 0 ;
	IF machine_standby=TRUE THEN
		xtrigger_control := TRUE;
	END_IF
ELSE
	standby_write := 1 ;
	IF machine_standby=FALSE THEN
		xtrigger_control := TRUE;
	END_IF	
END_IF


IF defrost_button THEN
	defrost_write := 1 ;
	IF defrost=FALSE THEN
		xtrigger_man_defrost := TRUE;
	END_IF
ELSE
	defrost_write := 0 ;

END_IF

// Door open timers
door_open_trigger(clk:=door_open);
door_close_trigger(clk:=door_open);

timer_door_open(IN:=timer_enable, PT:=T#30D);
timer_door_closed(IN:=timer2_enable, PT:=T#30D);

IF door_open_trigger.Q THEN
	closetime_tot := opentime_tot + timer_door_closed.ET;
	timer_enable := TRUE;
	timer2_enable := FALSE;
END_IF

IF door_close_trigger.Q THEN
	opentime_tot := opentime_tot + timer_door_open.ET;
	timer_enable := FALSE;
	timer2_enable := TRUE ;
END_IF


total_time := opentime_tot + closetime_tot ;

opentime_ms := TO_LREAL(TO_UDINT(opentime_tot) / 1000.0);
totaltime_ms := TO_LREAL(TO_UDINT(total_time) / 1000.0);

opentime_proc := (opentime_ms /totaltime_ms)*100 ;
IF resettimer_button THEN
	opentime_tot := T#0S ;
	closetime_tot := T#0S ;
	total_time := T#0S;
END_IF






// Graphic controls
IF select_trendvalue > 0 THEN
	show_trendvalue[select_trendvalue]:= TRUE;
ELSIF select_trendvalue = 0 THEN
	FOR i := 0 TO 50 DO
      show_trendvalue[i] := FALSE;
   	END_FOR
END_IF ;

END_PROGRAM

// Device/Application/Provision_4
PROGRAM Provision_4
VAR



modbus_var : ARRAY[0..800] OF WORD;
modbus_var1 : ARRAY[2000..2010] OF WORD;
timer_door_open : TON ;
timer_door_closed : TON ;
delay_timer : TON ;
open_time : TIME ;
total_time : TIME ;
opentime_tot : TIME ;
opentime_proc : REAL ;
closetime_tot : TIME ; 
{attribute 'ac_persist' := 'PersistenceChannel'}
set_delaytime : TIME := T#1S;
timer_enable : BOOL;
timer2_enable : BOOL;
timer_elapsed : BOOL ;
start_timer : BOOL := TRUE;
doorclose : F_TRIG;
resettimer_button :BOOL ;
totaltime_ms : LREAL ;
opentime_ms : LREAL ;

temp_provision_room : REAL;
temp_defrost : REAL;
regulator_temp : REAL;

set_point: REAL;
reg2 : REAL ;
reg3 : REAL ;
reg4 : REAL ;
reg5 : REAL ;
reg6 : REAL ;
reg7 : REAL ;
reg8 : REAL ;
reg9 : REAL ;
reg10 : WORD ;
reg11 : REAL ;
reg12 : REAL ;
reg13 : REAL ;
reg14 : REAL ;
reg15 : REAL ;
reg16 : REAL ;
reg17 : REAL ;
T1_offset : REAL ;
T2_offset : REAL ;
T3_offset : REAL ;
T1_span : REAL ;
T2_span : REAL ;
T3_span : REAL ;
valore_tasto1_V : REAL ;
valore_tasto_UP : REAL ;
valore_tasto_DW : REAL ;
valore_tasto_X : REAL ;
Test_display : REAL ;
Tasto_attualmente_premuto : REAL ;
Password : REAL ;

{attribute 'ac_persist' := 'PersistenceChannel'}
preset_parameters : REAL ;
preset_parameters_write_int :INT;
{attribute 'ac_persist' := 'PersistenceChannel'}
Readout_scale : REAL ;
{attribute 'ac_persist' := 'PersistenceChannel'}
Readout_scale_write_int : INT;
{attribute 'ac_persist' := 'PersistenceChannel'}
Minimum_temperature_setpoint : REAL ;
Minimum_temperature_setpoint_write_int : INT ;
{attribute 'ac_persist' := 'PersistenceChannel'}
Maximum_temperature_setpoint : REAL ;
Maximum_temperature_setpoint_write_int : INT ;
setp_write : REAL ;
{attribute 'ac_persist' := 'PersistenceChannel'}
Setpoint : REAL ;
{attribute 'ac_persist' := 'PersistenceChannel'}
Thermostat_OFF_ON_ref_to_SP : REAL  ;
{attribute 'ac_persist' := 'PersistenceChannel'}
Thermostat_ON_OFF_ref_to_SP : REAL  ;
Thermostat_OFF_ON_write : REAL  := 1.0 ;
Thermostat_ON_OFF_write : REAL  := 1.0 ;
Thermostat_OFF_ON_write_word : WORD ;
Thermostat_ON_OFF_write_word : WORD ;
Time_based_defrost_write : REAL   := 8.0  ;
Time_based_defrost_write_word : WORD  ;
Defrost_end_temperature_write : REAL  := 20.0 ;
Defrost_end_temperature_write_word : WORD ;
Fan_restart_temperature_after_defrost_write : REAL ;
Fan_restart_temperature_after_defrost_write_int : INT ;
Maximum_defrost_duration_write : REAL ;
Maximum_defrost_duration_write_word : WORD ;
defrost_write : WORD :=0 ;
{attribute 'ac_persist' := 'PersistenceChannel'}
CH_minimum_OFF_time : REAL ;
CH_minimum_OFF_time_write_int : INT ;
{attribute 'ac_persist' := 'PersistenceChannel'}
CH_minimum_ON_time : REAL ;
CH_minimum_ON_time_write_int : INT ;
{attribute 'ac_persist' := 'PersistenceChannel'}
CH_output_ON_when_probe_T1_is_faulty : REAL ;
CH_output_ON_when_probe_T1_is_faulty_write_int : INT ;
{attribute 'ac_persist' := 'PersistenceChannel'}
CH_output_OFF_when_probe_T1_is_faulty : REAL ;
CH_output_OFF_when_probe_T1_is_faulty_write_int : INT ;

{attribute 'ac_persist' := 'PersistenceChannel'}
Defrost_start_mode : REAL ;
{attribute 'ac_persist' := 'PersistenceChannel'}
Time_based_defrost : REAL ;
{attribute 'ac_persist' := 'PersistenceChannel'}
Minimum_Time_Between_Defrost : REAL ;
Minimum_Time_Between_Defrost_write_int : INT;
{attribute 'ac_persist' := 'PersistenceChannel'}
Defrost_time_optimization : REAL ;
Defrost_time_optimization_write_int : INT;
{attribute 'ac_persist' := 'PersistenceChannel'}
Defrost_type : REAL ;
Defrost_type_write_int : INT;
{attribute 'ac_persist' := 'PersistenceChannel'}
Delay_for_pressure_equalization_for_hot_gas : REAL ;
{attribute 'ac_persist' := 'PersistenceChannel'}
Defrost_end_temperature : REAL ;
{attribute 'ac_persist' := 'PersistenceChannel'}
Maximum_defrost_duration : REAL ;
{attribute 'ac_persist' := 'PersistenceChannel'}
Drain_down_time : REAL ;
Drain_down_time_write : REAL;
Drain_down_time_write_int : INT;
{attribute 'ac_persist' := 'PersistenceChannel'}
Display_defrost_mode : REAL ;
{attribute 'ac_persist' := 'PersistenceChannel'}
Display_delay : REAL ;
Display_delay_write_int : INT;
{attribute 'ac_persist' := 'PersistenceChannel'}
Fans_active_during_defrost : REAL ;
Fans_active_during_defrost_write_int : INT;
{attribute 'ac_persist' := 'PersistenceChannel'}
Fan_restart_temperature_after_defrost : REAL ;
{attribute 'ac_persist' := 'PersistenceChannel'}
Fan_stop_temperature : REAL ;
Fan_stop_temperature_write_int : INT ;
{attribute 'ac_persist' := 'PersistenceChannel'}
Maximum_fan_stop_for_FDD_FET : REAL ;
Maximum_fan_stop_for_FDD_FET_write_int : INT ;
{attribute 'ac_persist' := 'PersistenceChannel'}
Fan_mode_during_thermostatic_control : REAL ;
Fan_mode_during_thermostatic_control_write_int : INT ;
{attribute 'ac_persist' := 'PersistenceChannel'}
Target_evaporator_temperature : REAL ;
{attribute 'ac_persist' := 'PersistenceChannel'}
Fan_stop_delay_after_compressor_stop : REAL ;
{attribute 'ac_persist' := 'PersistenceChannel'}
Timed_fan_stop : REAL ;
{attribute 'ac_persist' := 'PersistenceChannel'}
Timed_fan_run : REAL ;
{attribute 'ac_persist' := 'PersistenceChannel'}
Fan_Minimum_Stop : REAL ;
{attribute 'ac_persist' := 'PersistenceChannel'}
Alarm_threshold_management : REAL ;
Alarm_threshold_management_write_int : INT ;
{attribute 'ac_persist' := 'PersistenceChannel'}
Low_temperature_alarm_threshold : REAL ;
{attribute 'ac_persist' := 'PersistenceChannel'}
High_temperature_alarm_threshold : REAL ;
Low_temperature_alarm_thres_write  : REAL := -20.0 ;
High_temperature_alarm_thres_write : REAL := 20.0 ;
Low_temperature_alarm_thres_write_word : WORD ;
High_temperature_alarm_thres_write_word : WORD ;
muteAlarm : WORD := 1;

{attribute 'ac_persist' := 'PersistenceChannel'}
Low_temperature_alarm_differential : REAL ;
{attribute 'ac_persist' := 'PersistenceChannel'}
High_temperature_alarm_differential : REAL ;
{attribute 'ac_persist' := 'PersistenceChannel'}
Probe_used_for_temperature_alarm_detection : REAL ;
{attribute 'ac_persist' := 'PersistenceChannel'}
Temperature_alarm_delay : REAL ;
Temperature_alarm_delay_write_int : INT ;
{attribute 'ac_persist' := 'PersistenceChannel'}
Operation_in_case_of_high_condenser_alarm : REAL ;
{attribute 'ac_persist' := 'PersistenceChannel'}
Condensation_temperature_alarm : REAL ;
{attribute 'ac_persist' := 'PersistenceChannel'}
Standby_button_enabling : REAL ;
{attribute 'ac_persist' := 'PersistenceChannel'}
Door_switch_input_mode : REAL ;
Door_switch_input_mode_write_int : INT ;
{attribute 'ac_persist' := 'PersistenceChannel'}
Door_alarm_delay : REAL ;
Door_alarm_delay_write_int : INT ;
{attribute 'ac_persist' := 'PersistenceChannel'}
Compressor_stop_delay : REAL ;
Compressor_stop_delay_write_int : INT ;
{attribute 'ac_persist' := 'PersistenceChannel'}
Door_stop_timeout : REAL ;
Door_stop_timeout_write_int : INT ;
{attribute 'ac_persist' := 'PersistenceChannel'}
DI1_digital_input_operation : REAL ;
{attribute 'ac_persist' := 'PersistenceChannel'}
DI1_digital_input_activation : REAL ;
{attribute 'ac_persist' := 'PersistenceChannel'}
DI2_digital_input_operation : REAL ;
{attribute 'ac_persist' := 'PersistenceChannel'}
DI2_digital_input_activation : REAL ;
DI1_digital_input_operation_write_int : INT ;
DI1_digital_input_activation_write_int : INT ;
DI2_digital_input_operation_write_int : INT ;
DI2_digital_input_activation_write_int : INT ;
{attribute 'ac_persist' := 'PersistenceChannel'}
Light_control_mode : REAL ;
Light_control_mode_write_int : INT ;
{attribute 'ac_persist' := 'PersistenceChannel'}
standby : REAL;
standby_write : INT;
{attribute 'ac_persist' := 'PersistenceChannel'}
Light_control : REAL;

write_data_alarm : R_TRIG;
write_data_setp : R_TRIG;
write_data_defrost : R_TRIG;
write_data_mute : R_TRIG;
write_data_control : R_TRIG;
write_data_man_defrost : R_TRIG;
door_open_trigger : R_TRIG ;
door_close_trigger : F_TRIG ;
set_param_trigger : R_TRIG ;
get_param_trigger : R_TRIG ;
all_param_read : BOOL ;
no_loop : INT :=0 ;


control_button : BOOL  := TRUE ;
defrost_button : BOOL  := FALSE ;
setpoint_button : BOOL ;
read_param_button : BOOL ;
{attribute 'ac_persist' := 'PersistenceChannel'}
RL1_output_operation : REAL ;
{attribute 'ac_persist' := 'PersistenceChannel'}
RL2_output_operation : REAL ;
{attribute 'ac_persist' := 'PersistenceChannel'}
RL3_output_operation : REAL ;
{attribute 'ac_persist' := 'PersistenceChannel'}
RL4_output_operation : REAL ;
RL1_output_operation_write_int : INT ;
RL2_output_operation_write_int : INT ;
RL3_output_operation_write_int : INT ;
RL4_output_operation_write_int : INT ;
{attribute 'ac_persist' := 'PersistenceChannel'}
Probe_T1_offset : REAL ;
{attribute 'ac_persist' := 'PersistenceChannel'}
Probe_T2_enable : REAL ;
{attribute 'ac_persist' := 'PersistenceChannel'}
Probe_T2_offset : REAL ;
{attribute 'ac_persist' := 'PersistenceChannel'}
Auxiliary_probe_T3_operation : REAL ;
{attribute 'ac_persist' := 'PersistenceChannel'}
Probe_T3_offset : REAL ;
{attribute 'ac_persist' := 'PersistenceChannel'}
Delay_for_minimum_and_maximum_temperature_logging : REAL ;
{attribute 'ac_persist' := 'PersistenceChannel'}
Selects_the_temperature_probe_to_be_displayed : REAL ;
{attribute 'ac_persist' := 'PersistenceChannel'}
The_relative_weight_of_T2_on_T1 : REAL ;
{attribute 'ac_persist' := 'PersistenceChannel'}
Display_slowdown : REAL ;
Display_slowdown_write_int : INT ;
{attribute 'ac_persist' := 'PersistenceChannel'}
Address_for_PC_communication : REAL ;
Address_for_PC_communication_write_int : INT ;
{attribute 'ac_persist' := 'PersistenceChannel'}
Modbus_protocol_selection : REAL ;
Modbus_protocol_selection_write_int : INT ;
// Word variables
Status_BITs_0_to_15 : WORD;
Status_BITs_16_to_31 : WORD;
Alarm_BITs_0_to_15 : WORD;
setp_write_word : WORD ;
Fan_stop_temperature_write_word : WORD ;

dig1 : BOOL;
dig2 : BOOL;
dout1 : BOOL;
dout2 : BOOL;
dout3 : BOOL;
dout4 : BOOL;
alarm : BOOL;
buzzer_mute : BOOL;
defrost : BOOL;
door_open : BOOL;
test : BOOL;
machine_standby : BOOL;
T1_failure  : BOOL;
T2_failure  : BOOL;
T3_failure  : BOOL;
Low_temperature  : BOOL;
High_temperature  : BOOL;
High_condenser_temperature  : BOOL;
Generic_alarm  : BOOL;
Door_open_alarm  : BOOL;
RL1 : BOOL;
RL2 : BOOL;
RL3 : BOOL;
SSR : BOOL;
deactivate_defrost_button : BOOL ;
modbus_communication : BOOL ;
comm_indicator : REAL ;



//triggers for writing setpoints and parameters
xtrigger_alarm : BOOL;
xtrigger_setp : BOOL;
xtrigger_defrost : BOOL;
xtrigger_mute : BOOL;
xtrigger_control : BOOL;
xtrigger_man_defrost : BOOL;
xtrigger_get_param : BOOL;
xtrigger_set_param : BOOL;








//Graphic variables
Unit_switch_status : INT;
i : INT;
show_trendvalue : ARRAY[0..50] OF BOOL;
select_trendvalue : INT :=0 ;

END_VAR




temp_provision_room:= scaleFunction(modbus_var[0],0.1, 0);
temp_defrost := scaleFunction(modbus_var[1],0.1, 0);
reg2 := scaleFunction(modbus_var[2],0.1, 0); // not used ?
reg3 := scaleFunction(modbus_var[3],0.1, 0); // not used ?
reg4 := scaleFunction(modbus_var[4],0.1, 0); // not used ?
reg5 := scaleFunction(modbus_var[5],0.1, 0); // not used ?
reg6 := scaleFunction(modbus_var[6],0.1, 0); // not used ?
reg7 := scaleFunction(modbus_var[7],0.1, 0); // not used ?
reg8 := scaleFunction(modbus_var[8],0.1, 0); // not used ?
reg9 := scaleFunction(modbus_var[9],0.1, 0); // not used ?
reg10 := modbus_var[10]; // not used ?
set_point := scaleFunction(modbus_var[11],0.1, 0);  // not used ?
reg12 := scaleFunction(modbus_var[12],0.1, 0); // not used ?
reg13 := scaleFunction(modbus_var[13],0.1, 0); // not used ?
reg14 := scaleFunction(modbus_var[14],0.1, 0); // not used ?
reg15 := scaleFunction(modbus_var[15],0.1, 0); // not used ?
reg16 := scaleFunction(modbus_var[16],0.1, 0); // not used ?
reg17 := scaleFunction(modbus_var[17],0.1, 0); // not used ?

// Non changeable parameters

T1_offset := scaleFunction(modbus_var1[2000],1, 0);
T2_offset := scaleFunction(modbus_var1[2001],1, 2);
T3_offset := scaleFunction(modbus_var1[2002],1, 3);
T1_span := scaleFunction(modbus_var1[2003],1, 4);
T2_span := scaleFunction(modbus_var1[2004],1, 5);
T3_span := scaleFunction(modbus_var1[2005],1, 6);

valore_tasto1_V := scaleFunction(modbus_var[150],1, 6);
valore_tasto_UP := scaleFunction(modbus_var[151],1, 6);
valore_tasto_DW := scaleFunction(modbus_var[152],1, 6);
valore_tasto_X := scaleFunction(modbus_var[153],1, 6);

Test_display := scaleFunction(modbus_var[193],1, 0);
Tasto_attualmente_premuto := scaleFunction(modbus_var[194],1, 0);
Password := scaleFunction(modbus_var[197],1, 0);

preset_parameters:= scaleFunction(modbus_var[200],1, 0);

Setpoint:= scaleFunction(modbus_var[303],0.1, 0);
Thermostat_OFF_ON_ref_to_SP:= scaleFunction(modbus_var[304],0.1, 0);
Thermostat_ON_OFF_ref_to_SP:= scaleFunction(modbus_var[305],0.1, 0);

Defrost_start_mode:= scaleFunction(modbus_var[400],1, 0);
Time_based_defrost:= scaleFunction(modbus_var[401],1, 0);

Delay_for_pressure_equalization_for_hot_gas:= scaleFunction(modbus_var[405],1, 0);

Defrost_end_temperature:= scaleFunction(modbus_var[406],0.1, 0);
Maximum_defrost_duration:= scaleFunction(modbus_var[407],1, 0);

Drain_down_time:= scaleFunction(modbus_var[408],1, 0);
Display_defrost_mode:= scaleFunction(modbus_var[409],1, 0);

Target_evaporator_temperature:= scaleFunction(modbus_var[453],0.1, 0);
Fan_stop_delay_after_compressor_stop:= scaleFunction(modbus_var[454],1, 0);
Timed_fan_stop:= scaleFunction(modbus_var[455],1, 0);
Timed_fan_run:= scaleFunction(modbus_var[456],1, 0);
Fan_Minimum_Stop:= scaleFunction(modbus_var[457],1, 0);


Low_temperature_alarm_threshold:= scaleFunction(modbus_var[501],0.1, 0);
High_temperature_alarm_threshold:= scaleFunction(modbus_var[502],0.1, 0);
Low_temperature_alarm_differential:= scaleFunction(modbus_var[503],0.1, 0);
High_temperature_alarm_differential:= scaleFunction(modbus_var[504],0.1, 0);
Probe_used_for_temperature_alarm_detection:= scaleFunction(modbus_var[505],1, 0);
Operation_in_case_of_high_condenser_alarm:= scaleFunction(modbus_var[507],1, 0);
Condensation_temperature_alarm:= scaleFunction(modbus_var[508],0.1, 0);

Standby_button_enabling:= scaleFunction(modbus_var[600],1, 0);



// Changeable parameters
delay_timer(IN:=read_param_button, PT:=set_delaytime);
IF read_param_button THEN
	Display_slowdown:= scaleFunction(modbus_var[208],1, 0);
	Readout_scale:= scaleFunction(modbus_var[300],1, 0);
	Minimum_temperature_setpoint:= scaleFunction(modbus_var[301],0.1, 0);
	Maximum_temperature_setpoint:= scaleFunction(modbus_var[302],0.1, 0);
	CH_minimum_OFF_time:= scaleFunction(modbus_var[306],1, 0);
	CH_minimum_ON_time:= scaleFunction(modbus_var[307],1, 0);
	CH_output_ON_when_probe_T1_is_faulty:= scaleFunction(modbus_var[308],1, 0);
	CH_output_OFF_when_probe_T1_is_faulty:= scaleFunction(modbus_var[309],1, 0);
	Minimum_Time_Between_Defrost:= scaleFunction(modbus_var[402],1, 0);
	Defrost_time_optimization:= scaleFunction(modbus_var[403],1, 0);
	Defrost_type:= scaleFunction(modbus_var[404],1, 0);
//	Defrost_end_temperature:= scaleFunction(modbus_var[406],1, 0);
//	Maximum_defrost_duration:= scaleFunction(modbus_var[407],1, 0);
	Display_delay:= scaleFunction(modbus_var[410],1, 0);
	Fans_active_during_defrost:= scaleFunction(modbus_var[411],1, 0);
	Fan_restart_temperature_after_defrost:= scaleFunction(modbus_var[412],0.1, 0);
	Fan_mode_during_thermostatic_control:= scaleFunction(modbus_var[452],1, 0);
	Fan_stop_temperature:= scaleFunction(modbus_var[450],0.1, 0);
	Maximum_fan_stop_for_FDD_FET:= scaleFunction(modbus_var[451],1, 0);
	Alarm_threshold_management:= scaleFunction(modbus_var[500],1, 0);
	Temperature_alarm_delay:= scaleFunction(modbus_var[506],1, 0);
	Door_switch_input_mode:= scaleFunction(modbus_var[601],1, 0);
	Door_alarm_delay:= scaleFunction(modbus_var[602],1, 0);
	Compressor_stop_delay:= scaleFunction(modbus_var[603],1, 0);
	Door_stop_timeout:= scaleFunction(modbus_var[604],1, 0);
	DI1_digital_input_operation:= scaleFunction(modbus_var[605],1, 0);
	DI1_digital_input_activation:= scaleFunction(modbus_var[606],1, 0);
	DI2_digital_input_operation:= scaleFunction(modbus_var[607],1, 0);
	DI2_digital_input_activation:= scaleFunction(modbus_var[608],1, 0);
	Light_control_mode:= scaleFunction(modbus_var[609],1, 0);
	RL1_output_operation:= scaleFunction(modbus_var[650],1, 0);
	RL2_output_operation:= scaleFunction(modbus_var[651],1, 0);
	RL3_output_operation:= scaleFunction(modbus_var[652],1, 0);
	RL4_output_operation:= scaleFunction(modbus_var[653],1, 0);

	// no_loop :=no_loop +1 ;
	IF delay_timer.Q THEN
		read_param_button := FALSE ;
		no_loop:=0;
	END_IF	
END_IF










standby:= scaleFunction(modbus_var[702],1, 0);
Light_control:= scaleFunction(modbus_var[703],1, 0);




Probe_T1_offset:= scaleFunction(modbus_var[201],0.1, 0);
Probe_T2_enable:= scaleFunction(modbus_var[202],1, 0);
Probe_T2_offset:= scaleFunction(modbus_var[203],0.1, 0);
Auxiliary_probe_T3_operation:= scaleFunction(modbus_var[204],1, 0);
Probe_T3_offset:= scaleFunction(modbus_var[205],0.1, 0);
Selects_the_temperature_probe_to_be_displayed:= scaleFunction(modbus_var[206],1, 0);
The_relative_weight_of_T2_on_T1:= scaleFunction(modbus_var[207],1, 0);

Address_for_PC_communication:= scaleFunction(modbus_var[209],1, 0);
Modbus_protocol_selection:= scaleFunction(modbus_var[210],1, 0);
Delay_for_minimum_and_maximum_temperature_logging:= scaleFunction(modbus_var[211],1, 0);

//  Statusbits
Status_BITs_0_to_15 := modbus_var[100];
Status_BITs_16_to_31 := modbus_var[102];
Alarm_BITs_0_to_15 := modbus_var[101];


alarm := maskbitFunction(Status_BITs_0_to_15,0) OR NOT modbus_communication ;
buzzer_mute := maskbitFunction(Status_BITs_0_to_15,1);
defrost:= maskbitFunction(Status_BITs_0_to_15,2);
door_open := maskbitFunction(Status_BITs_0_to_15,3);
test := maskbitFunction(Status_BITs_0_to_15,4);
machine_standby := maskbitFunction(Status_BITs_0_to_15,5);


T1_failure := maskbitFunction(Alarm_BITs_0_to_15,0);
T2_failure := maskbitFunction(Alarm_BITs_0_to_15,1);
T3_failure := maskbitFunction(Alarm_BITs_0_to_15,2);
Low_temperature := maskbitFunction(Alarm_BITs_0_to_15,3);
High_temperature := maskbitFunction(Alarm_BITs_0_to_15,4);
High_condenser_temperature := maskbitFunction(Alarm_BITs_0_to_15,5);
Generic_alarm := maskbitFunction(Alarm_BITs_0_to_15,6);
Door_open_alarm := maskbitFunction(Alarm_BITs_0_to_15,7);

dout1 := maskbitFunction(Status_BITs_16_to_31,0); 
dout2 := maskbitFunction(Status_BITs_16_to_31,1);
dout3 := maskbitFunction(Status_BITs_16_to_31,2);
dout4 := maskbitFunction(Status_BITs_16_to_31,3);

RL1 := maskbitFunction(modbus_var[196],0);
RL2 := maskbitFunction(modbus_var[196],1);

RL3 := maskbitFunction(modbus_var[196],2);
SSR := maskbitFunction(modbus_var[196],3);


dig1 := maskbitFunction(reg10,0);
dig2 := maskbitFunction(reg10,1);

// Communication fault
comm_indicator := temp_provision_room + temp_defrost + reg2 + reg3 + reg4 + reg5
+ reg6 + reg7 + reg8 + reg9 + reg10 ;
IF comm_indicator = 0 THEN
	modbus_communication := FALSE ;
ELSE
	modbus_communication := TRUE ;
END_IF
	



// Parameter write values

setp_write_word := REAL_TO_INT(setp_write*10) ;
Thermostat_OFF_ON_write_word := REAL_TO_INT(Thermostat_OFF_ON_write*10) ;
Thermostat_ON_OFF_write_word:= REAL_TO_INT(Thermostat_ON_OFF_write*10) ;
Low_temperature_alarm_thres_write_word:= REAL_TO_INT(Low_temperature_alarm_thres_write*10);
High_temperature_alarm_thres_write_word:= REAL_TO_INT(High_temperature_alarm_thres_write*10);
muteAlarm :=1 ;
Time_based_defrost_write_word:= REAL_TO_INT(Time_based_defrost_write*1);
Defrost_end_temperature_write_word:= REAL_TO_INT(Defrost_end_temperature_write*10);
Drain_down_time_write_int:= REAL_TO_INT(Drain_down_time_write);
Maximum_defrost_duration_write_word:= REAL_TO_INT(Maximum_defrost_duration_write*1);
Fan_stop_temperature_write_word:= REAL_TO_INT(Fan_stop_temperature*10);
preset_parameters_write_int:=REAL_TO_INT(preset_parameters);
Readout_scale_write_int:=REAL_TO_INT(Readout_scale);
Minimum_temperature_setpoint_write_int:=REAL_TO_INT(Minimum_temperature_setpoint*10);
Maximum_temperature_setpoint_write_int:=REAL_TO_INT(Maximum_temperature_setpoint*10);
CH_minimum_OFF_time_write_int:=REAL_TO_INT(CH_minimum_OFF_time);
CH_minimum_ON_time_write_int:=REAL_TO_INT(CH_minimum_ON_time);
CH_output_ON_when_probe_T1_is_faulty_write_int:=REAL_TO_INT(CH_output_ON_when_probe_T1_is_faulty);
CH_output_OFF_when_probe_T1_is_faulty_write_int:=REAL_TO_INT(CH_output_OFF_when_probe_T1_is_faulty);
Minimum_Time_Between_Defrost_write_int:=REAL_TO_INT(Minimum_Time_Between_Defrost);
Defrost_time_optimization_write_int:=REAL_TO_INT(Defrost_time_optimization);
Defrost_type_write_int:=REAL_TO_INT(Defrost_type);
Display_delay_write_int:=REAL_TO_INT(Display_delay);
Fans_active_during_defrost_write_int:=REAL_TO_INT(Fans_active_during_defrost);
Fan_restart_temperature_after_defrost_write_int:=REAL_TO_INT(Fan_restart_temperature_after_defrost*10);
// Fan_stop_temperature_write_int:=REAL_TO_INT(Fan_stop_temperature);
Maximum_fan_stop_for_FDD_FET_write_int:=REAL_TO_INT(Maximum_fan_stop_for_FDD_FET);
Fan_mode_during_thermostatic_control_write_int:=REAL_TO_INT(Fan_mode_during_thermostatic_control);
Alarm_threshold_management_write_int:=REAL_TO_INT(Alarm_threshold_management);
Temperature_alarm_delay_write_int:=REAL_TO_INT(Temperature_alarm_delay);
Door_switch_input_mode_write_int:=REAL_TO_INT(Door_switch_input_mode);
Door_alarm_delay_write_int:=REAL_TO_INT(Door_alarm_delay);
Compressor_stop_delay_write_int:=REAL_TO_INT(Compressor_stop_delay);
Door_stop_timeout_write_int:=REAL_TO_INT(Door_stop_timeout);
DI1_digital_input_operation_write_int:=REAL_TO_INT(DI1_digital_input_operation);
DI1_digital_input_activation_write_int:=REAL_TO_INT(DI1_digital_input_activation);
DI2_digital_input_operation_write_int:=REAL_TO_INT(DI2_digital_input_operation);
DI2_digital_input_activation_write_int:=REAL_TO_INT(DI2_digital_input_activation);
Light_control_mode_write_int:=REAL_TO_INT(Light_control_mode);
RL1_output_operation_write_int:=REAL_TO_INT(RL1_output_operation);
RL2_output_operation_write_int:=REAL_TO_INT(RL2_output_operation);
RL3_output_operation_write_int:=REAL_TO_INT(RL3_output_operation);
RL4_output_operation_write_int:=REAL_TO_INT(RL4_output_operation);
Display_slowdown_write_int:=REAL_TO_INT(Display_slowdown);
Address_for_PC_communication_write_int:=REAL_TO_INT(Address_for_PC_communication);
Modbus_protocol_selection_write_int:=REAL_TO_INT(Modbus_protocol_selection);

write_data_alarm(clk:=xtrigger_alarm);
write_data_setp(clk:=xtrigger_setp);
write_data_defrost(clk:=xtrigger_defrost);
write_data_mute(clk:=xtrigger_mute);
write_data_control(clk:=xtrigger_control);
write_data_man_defrost(clk:=xtrigger_man_defrost);
get_param_trigger(clk:=xtrigger_get_param);
set_param_trigger(clk:=xtrigger_set_param);


IF control_button THEN
	standby_write := 0 ;
	IF machine_standby=TRUE THEN
		xtrigger_control := TRUE;
	END_IF
ELSE
	standby_write := 1 ;
	IF machine_standby=FALSE THEN
		xtrigger_control := TRUE;
	END_IF	
END_IF


IF defrost_button THEN
	defrost_write := 1 ;
	IF defrost=FALSE THEN
		xtrigger_man_defrost := TRUE;
	END_IF
ELSE
	defrost_write := 0 ;

END_IF

// Door open timers
door_open_trigger(clk:=door_open);
door_close_trigger(clk:=door_open);

timer_door_open(IN:=timer_enable, PT:=T#30D);
timer_door_closed(IN:=timer2_enable, PT:=T#30D);

IF door_open_trigger.Q THEN
	closetime_tot := opentime_tot + timer_door_closed.ET;
	timer_enable := TRUE;
	timer2_enable := FALSE;
END_IF

IF door_close_trigger.Q THEN
	opentime_tot := opentime_tot + timer_door_open.ET;
	timer_enable := FALSE;
	timer2_enable := TRUE ;
END_IF


total_time := opentime_tot + closetime_tot ;

opentime_ms := TO_LREAL(TO_UDINT(opentime_tot) / 1000.0);
totaltime_ms := TO_LREAL(TO_UDINT(total_time) / 1000.0);

opentime_proc := (opentime_ms /totaltime_ms)*100 ;
IF resettimer_button THEN
	opentime_tot := T#0S ;
	closetime_tot := T#0S ;
	total_time := T#0S;
END_IF






// Graphic controls
IF select_trendvalue > 0 THEN
	show_trendvalue[select_trendvalue]:= TRUE;
ELSIF select_trendvalue = 0 THEN
	FOR i := 0 TO 50 DO
      show_trendvalue[i] := FALSE;
   	END_FOR
END_IF ;

END_PROGRAM

// Device/Application/MainVisualization
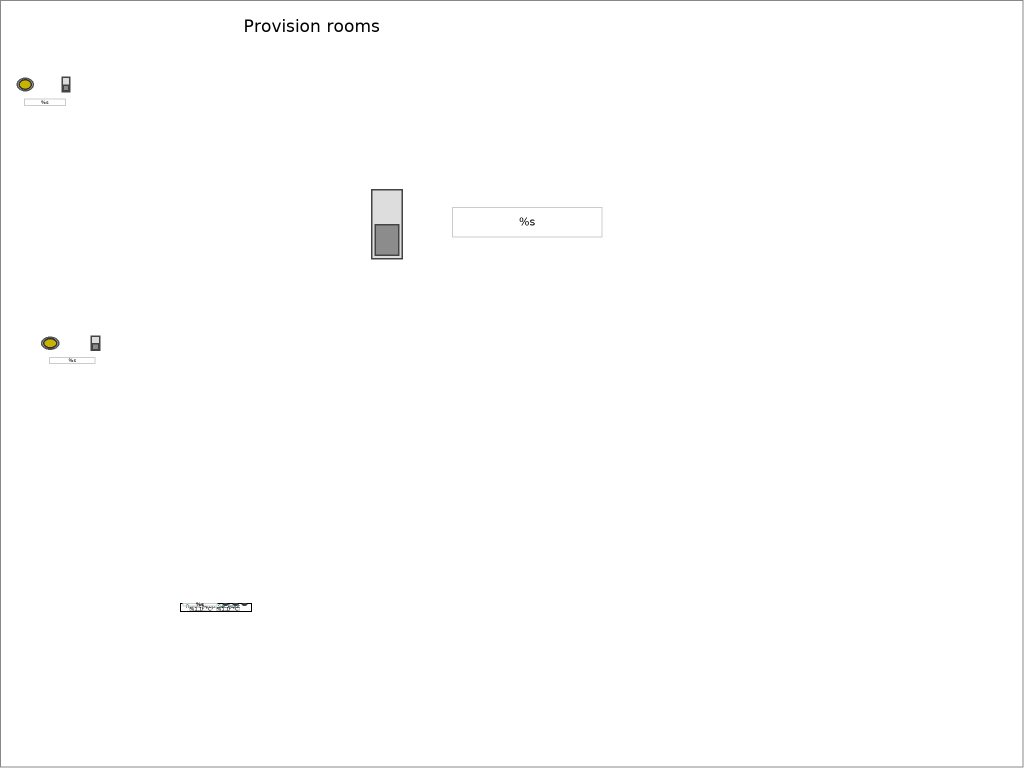
VISUALIZATION MainVisualization  // 1024x768
    Label (237,11 150x30), "Provision rooms"
    Frame (-2,69 282x168)
        shows objectvisiu(provroom := Main_program.Prov1)
    Frame (20,328 313x165)
        shows objectvisiu(provroom := Main_program.Prov2)
    DipSwitch (352,189 70x70), variable: Main_program.status_switch, behaviour: TOGGLE, style: Switch-DipSwitch-Gray
    Textfield (452,207 150x30), "%s", text variable: Main_program.text_message
    Frame (179,602 273x86)
        shows ProvRoomTemp(provroomTemp := Main_program.Provision_room1)
END_VISUALIZATION

// Device/Application/objectvisiu
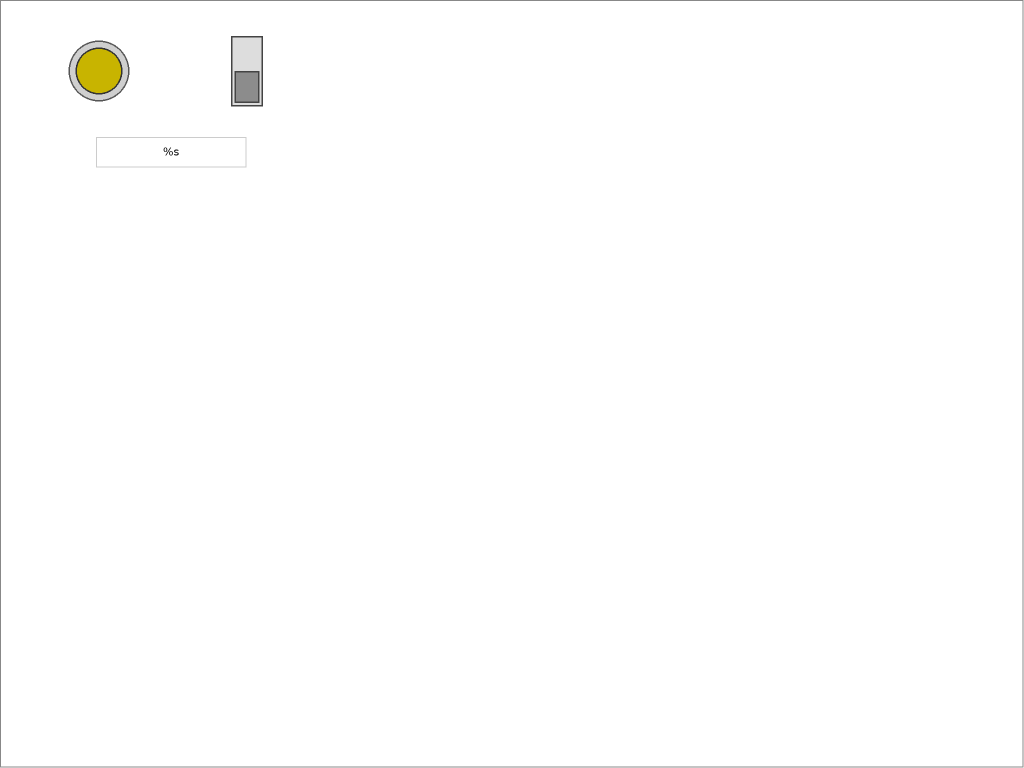
VISUALIZATION objectvisiu  // 1024x768
VAR_IN_OUT
	provroom : clsLampFunction();
END_VAR
    Lamp1 (64,36 70x70), variable: provroom.Lamp, style: Lamp-Lamp1-Yellow
    DipSwitch (212,36 70x70), variable: provroom.xSwitch, behaviour: TOGGLE, style: Switch-DipSwitch-Gray
        OnValueChanged:  ToggleVariable=provroom.Switch
    Textfield (96,137 150x30), "%s", text variable: provroom.Value
END_VISUALIZATION

// Device/Application/Provision_1_2_3_SysOverview
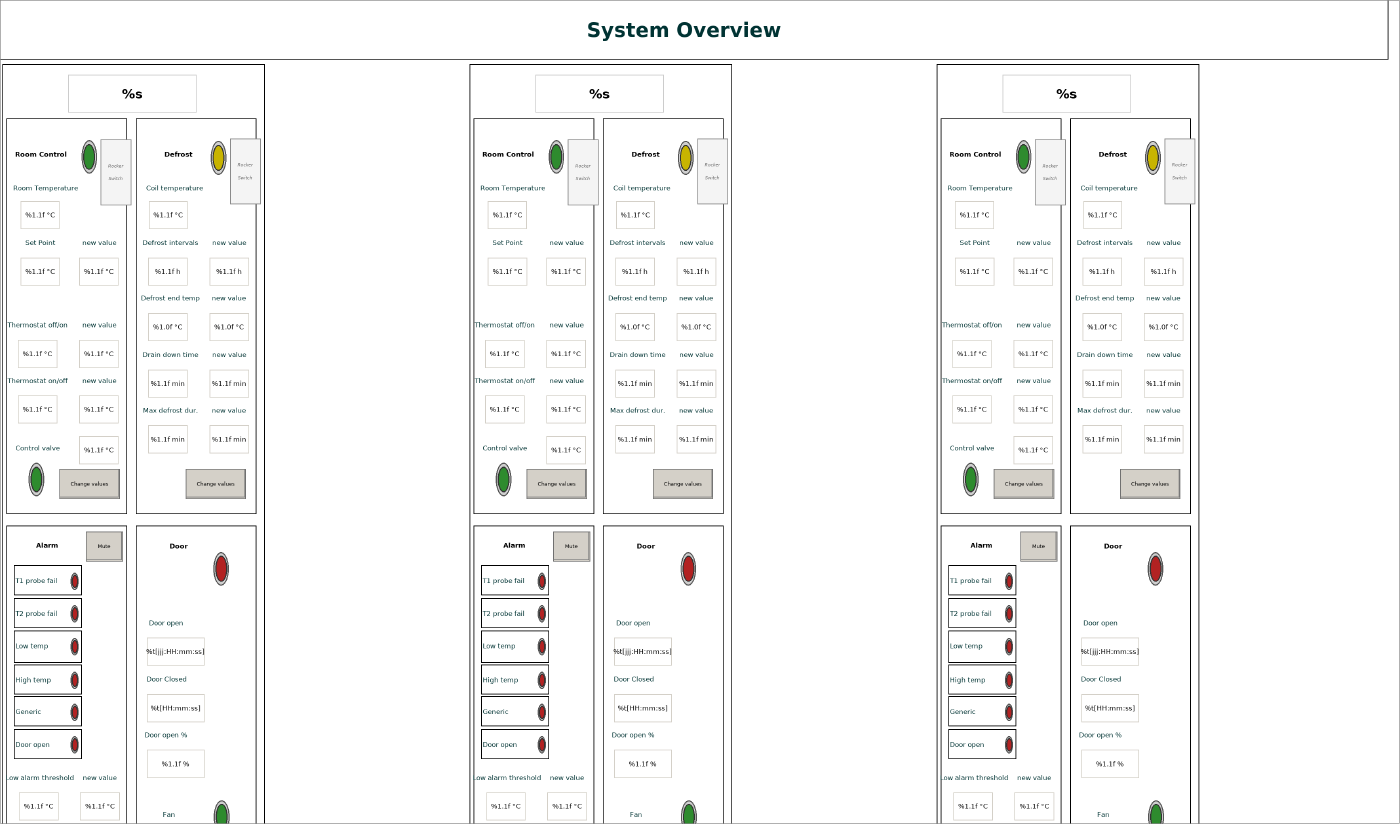
VISUALIZATION Provision_1_2_3_SysOverview  // 1768x1041
    Rectangle (0,0 1753x75)
    Label (456,1 816x73), "System Overview"
    Frame (3,76 583x963)
        shows ProvRoom_All(provroomTemp := Main_program.Provision_room1)
    Frame (593,76 583x963)
        shows ProvRoom_All(provroomTemp := Main_program.Provision_room2)
    Frame (1183,76 583x963)
        shows ProvRoom_All(provroomTemp := Main_program.Provision_room3)
END_VISUALIZATION

// Device/Application/Provision_1_Values
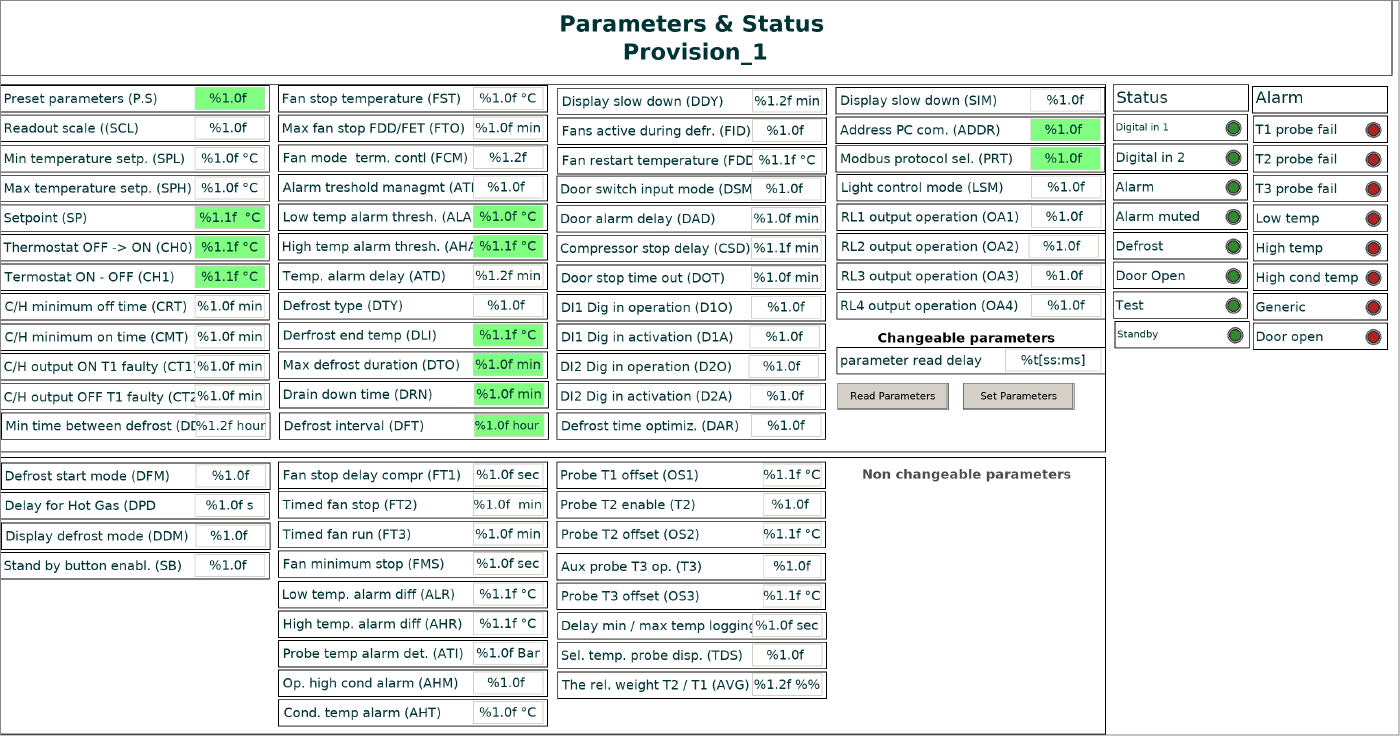
VISUALIZATION Provision_1_Values  // 1560x821
    Rectangle (0,94 1232x410)
    Rectangle (0,510 1232x309)
    Rectangle (0,0 1551x84)
    Label (319,7 912x70), "Parameters & Status Provision_1"
    Rectangle (0,95 300x30)
    Label (1,90 208x40), "Preset parameters (P.S)"
    Textfield (217,97 78x25), "%1.0f", tooltip "Provision_1.preset_parameters", text variable: Provision_1.preset_parameters
        p4168582468: Provision_1.preset_parameters
        OnMouseClick: write the text variable via Default
    Rectangle (0,128 300x30)
    Label (1,123 209x40), "Readout scale ((SCL)"
    Textfield (217,130 78x25), "%1.0f", tooltip "Provision_1.Readout_scale", text variable: Provision_1.Readout_scale
        p4168582468: Provision_1.Readout_scale
        OnMouseClick: write the text variable via Default
    Rectangle (0,162 300x30)
    Label (1,157 211x40), "Min temperature setp. (SPL)"
    Textfield (217,164 78x25), "%1.0f °C", tooltip "Provision_1.Minimum_temperature_setpoint", text variable: Provision_1.Minimum_temperature_setpoint
        p4168582468: Provision_1.Minimum_temperature_setpoint
        OnMouseClick: write the text variable via Default
    Rectangle (0,195 300x30)
    Label (1,190 216x40), "Max temperature setp. (SPH)"
    Textfield (217,197 78x25), "%1.0f °C", tooltip "Provision_1.Maximum_temperature_setpoint", text variable: Provision_1.Maximum_temperature_setpoint
        p4168582468: Provision_1.Maximum_temperature_setpoint
        OnMouseClick: write the text variable via Default
    Rectangle (310,95 300x30)
    Label (311,90 209x40), "Fan stop temperature (FST)"
    Textfield (527,97 78x25), "%1.0f °C", tooltip "Provision_1.Fan_stop_temperature", text variable: Provision_1.Fan_stop_temperature
        p4168582468: Provision_1.Fan_stop_temperature
        OnMouseClick: write the text variable via Default
    Rectangle (310,128 300x30)
    Label (311,123 204x40), "Max fan stop FDD/FET (FTO)"
    Textfield (527,130 78x25), "%1.0f min", tooltip "Provision_1.Maximum_fan_stop_for_FDD_FET", text variable: Provision_1.Maximum_fan_stop_for_FDD_FET
        p4168582468: Provision_1.Maximum_fan_stop_for_FDD_FET
        OnMouseClick: write the text variable via Default
    Rectangle (310,161 300x30)
    Label (312,156 209x40), "Fan mode term. contl (FCM)"
    Textfield (527,163 78x25), "%1.2f", tooltip "Provision_1.Fan_mode_during_thermostatic_control", text variable: Provision_1.Fan_mode_during_thermostatic_control
        p4168582468: Provision_1.Fan_mode_during_thermostatic_control
        OnMouseClick: write the text variable via Default
    Rectangle (310,542 300x30)
    Label (312,538 214x40), "Target evaporator temp. (FET)"
    Textfield (527,544 78x25), "%1.0f °C", tooltip "Provision_1.Timed_fan_stop", text variable: Provision_1.Timed_fan_stop
        p4168582468: Provision_1.Timed_fan_stop
    Rectangle (310,515 300x30)
    Label (312,510 216x40), "Fan stop delay compr (FT1)"
    Textfield (527,517 78x25), "%1.0f sec", tooltip "Provision_1.Fan_stop_delay_after_compressor_stop", text variable: Provision_1.Fan_stop_delay_after_compressor_stop
        p4168582468: Provision_1.Fan_stop_delay_after_compressor_stop
    Rectangle (310,548 300x30)
    Label (312,543 215x40), "Timed fan stop (FT2)"
    Textfield (527,550 78x25), "%1.0f min", tooltip "Provision_1.Timed_fan_stop", text variable: Provision_1.Timed_fan_stop
        p4168582468: Provision_1.Timed_fan_stop
    Rectangle (310,581 300x30)
    Label (312,576 218x40), "Timed fan run (FT3)"
    Textfield (527,583 78x25), "%1.0f min", tooltip "Provision_1.Timed_fan_run", text variable: Provision_1.Timed_fan_run
        p4168582468: Provision_1.Timed_fan_run
    Rectangle (310,614 300x30)
    Label (312,609 214x40), "Fan minimum stop (FMS)"
    Textfield (527,616 78x25), "%1.0f sec", tooltip "Provision_1.Fan_Minimum_Stop", text variable: Provision_1.Fan_Minimum_Stop
        p4168582468: Provision_1.Fan_Minimum_Stop
    Rectangle (310,194 300x30)
    Label (312,189 216x40), "Alarm treshold managmt (ATM)"
    Textfield (527,196 78x25), "%1.0f", tooltip "Provision_1.Alarm_threshold_management", text variable: Provision_1.Alarm_threshold_management
        p4168582468: Provision_1.Alarm_threshold_management
        OnMouseClick: write the text variable via Default
    Rectangle (620,515 300x30)
    Label (621,514 174x32), "Probe T1 offset (OS1)"
    Textfield (850,517 65x25), "%1.1f °C", tooltip "Provision_1.Probe_T1_offset", text variable: Provision_1.Probe_T1_offset
        p4168582468: Provision_1.Probe_T1_offset
    Rectangle (620,548 300x30)
    Label (621,547 173x32), "Probe T2 enable (T2)"
    Textfield (850,550 65x25), "%1.0f", tooltip "Provision_1.Probe_T2_enable", text variable: Provision_1.Probe_T2_enable
        p4168582468: Provision_1.Probe_T2_enable
    Rectangle (620,617 300x30)
    Label (622,616 177x32), "Aux probe T3 op. (T3)"
    Textfield (850,619 65x25), "%1.0f", tooltip "Provision_1.Auxiliary_probe_T3_operation", text variable: Provision_1.Auxiliary_probe_T3_operation
        p4168582468: Provision_1.Auxiliary_probe_T3_operation
    Rectangle (620,650 300x30)
    Label (622,651 177x28), "Probe T3 offset (OS3)"
    Textfield (850,652 65x25), "%1.1f °C", tooltip "Provision_1.Probe_T3_offset", text variable: Provision_1.Probe_T3_offset
        p4168582468: Provision_1.Probe_T3_offset
    Rectangle (0,228 300x30)
    Label (1,223 213x40), "Setpoint (SP)"
    Textfield (217,230 78x25), "%1.1f °C", tooltip "Provision_1.Setpoint", text variable: Provision_1.Setpoint
        p4168582468: Provision_1.Setpoint
        OnMouseClick: write the text variable via Default
    Rectangle (0,261 300x30)
    Label (1,256 214x40), "Thermostat OFF -> ON (CH0)"
    Textfield (217,263 78x25), "%1.1f °C", tooltip "Provision_1.Thermostat_OFF_ON_ref_to_SP", text variable: Provision_1.Thermostat_OFF_ON_ref_to_SP
        p4168582468: Provision_1.Thermostat_OFF_ON_ref_to_SP
        OnMouseClick: write the text variable via Default
    Rectangle (0,294 300x30)
    Label (2,289 213x40), "Termostat ON - OFF (CH1)"
    Textfield (217,296 78x25), "%1.1f °C", tooltip "Provision_1.Thermostat_ON_OFF_ref_to_SP", text variable: Provision_1.Thermostat_ON_OFF_ref_to_SP
        p4168582468: Provision_1.Thermostat_ON_OFF_ref_to_SP
        OnMouseClick: write the text variable via Default
    Rectangle (0,361 300x30)
    Textfield (217,363 78x25), "%1.0f min", tooltip "Provision_1.CH_minimum_ON_time", text variable: Provision_1.CH_minimum_ON_time
        p4168582468: Provision_1.CH_minimum_ON_time
        OnMouseClick: write the text variable via Default
    Rectangle (0,327 300x30)
    Label (2,322 212x40), "C/H minimum off time (CRT)"
    Textfield (217,329 78x25), "%1.0f min", tooltip "Provision_1.CH_minimum_OFF_time", text variable: Provision_1.CH_minimum_OFF_time
        p4168582468: Provision_1.CH_minimum_OFF_time
        OnMouseClick: write the text variable via Default
    Label (2,356 210x40), "C/H minimum on time (CMT)"
    Rectangle (620,581 300x30)
    Label (622,580 174x32), "Probe T2 offset (OS2)"
    Textfield (850,583 65x25), "%1.1f °C", tooltip "Provision_1.Probe_T2_offset", text variable: Provision_1.Probe_T2_offset
        p4168582468: Provision_1.Probe_T2_offset
    Rectangle (0,616 300x30)
    Label (1,611 209x40), "Stand by button enabl. (SB)"
    Textfield (217,618 78x25), "%1.0f", tooltip "Provision_1.Standby_button_enabling", text variable: Provision_1.Standby_button_enabling
        p4168582468: Provision_1.Standby_button_enabling
    Rectangle (620,262 300x30)
    Label (621,257 210x40), "Compressor stop delay (CSD)"
    Textfield (837,264 78x25), "%1.1f min", tooltip "Provision_1.Compressor_stop_delay", text variable: Provision_1.Compressor_stop_delay
        p4168582468: Provision_1.Compressor_stop_delay
        OnMouseClick: write the text variable via Default
    Rectangle (620,295 300x30)
    Label (622,290 204x40), "Door stop time out (DOT)"
    Textfield (837,297 78x25), "%1.0f min", tooltip "Provision_1.Door_stop_timeout", text variable: Provision_1.Door_stop_timeout
        p4168582468: Provision_1.Door_stop_timeout
        OnMouseClick: write the text variable via Default
    Rectangle (620,328 300x30)
    Label (622,323 206x40), "DI1 Dig in operation (D1O)"
    Textfield (837,330 78x25), "%1.0f", tooltip "Provision_1.DI1_digital_input_operation", text variable: Provision_1.DI1_digital_input_operation
        p4168582468: Provision_1.DI1_digital_input_operation
        OnMouseClick: write the text variable via Default
    Rectangle (620,361 300x30)
    Label (622,356 216x40), "DI1 Dig in activation (D1A)"
    Textfield (835,363 78x25), "%1.0f", tooltip "Provision_1.DI1_digital_input_activation", text variable: Provision_1.DI1_digital_input_activation
        p4168582468: Provision_1.DI1_digital_input_activation
        OnMouseClick: write the text variable via Default
    Rectangle (620,394 300x30)
    Label (621,389 218x40), "DI2 Dig in operation (D2O)"
    Textfield (834,396 78x25), "%1.0f", tooltip "Provision_1.DI2_digital_input_operation", text variable: Provision_1.DI2_digital_input_operation
        p4168582468: Provision_1.DI2_digital_input_operation
        OnMouseClick: write the text variable via Default
    Rectangle (620,427 300x30)
    Label (621,422 215x40), "DI2 Dig in activation (D2A)"
    Textfield (836,429 78x25), "%1.0f", tooltip "Provision_1.DI2_digital_input_activation", text variable: Provision_1.DI2_digital_input_activation
        p4168582468: Provision_1.DI2_digital_input_activation
        OnMouseClick: write the text variable via Default
    Rectangle (932,194 300x30)
    Label (934,189 215x40), "Light control mode (LSM)"
    Textfield (1149,196 78x25), "%1.0f", tooltip "Provision_1.Light_control_mode", text variable: Provision_1.Light_control_mode
        p4168582468: Provision_1.Light_control_mode
        OnMouseClick: write the text variable via Default
    Rectangle (932,227 300x30)
    Label (934,222 210x40), "RL1 output operation (OA1)"
    Textfield (1149,229 78x25), "%1.0f", tooltip "Provision_1.RL1_output_operation", text variable: Provision_1.RL1_output_operation
        p4168582468: Provision_1.RL1_output_operation
        OnMouseClick: write the text variable via Default
    Rectangle (932,260 300x30)
    Label (934,255 214x40), "RL2 output operation (OA2)"
    Textfield (1146,262 78x25), "%1.0f", tooltip "Provision_1.RL2_output_operation", text variable: Provision_1.RL2_output_operation
        p4168582468: Provision_1.RL2_output_operation
        OnMouseClick: write the text variable via Default
    Rectangle (932,293 300x30)
    Label (934,288 207x40), "RL3 output operation (OA3)"
    Textfield (1149,295 78x25), "%1.0f", tooltip "Provision_1.RL3_output_operation", text variable: Provision_1.RL3_output_operation
        p4168582468: Provision_1.RL3_output_operation
        OnMouseClick: write the text variable via Default
    Rectangle (310,260 300x30)
    Label (311,255 204x40), "High temp alarm thresh. (AHA)"
    Textfield (527,262 78x25), "%1.1f °C", tooltip "Provision_1.High_temperature_alarm_threshold", text variable: Provision_1.High_temperature_alarm_threshold
        p4168582468: Provision_1.High_temperature_alarm_threshold
        OnMouseClick: write the text variable via Default
    Rectangle (310,648 300x30)
    Label (311,643 209x40), "Low temp. alarm diff (ALR)"
    Textfield (527,650 78x25), "%1.1f °C", tooltip "Provision_1.Low_temperature_alarm_differential", text variable: Provision_1.Low_temperature_alarm_differential
        p4168582468: Provision_1.Low_temperature_alarm_differential
    Rectangle (310,681 300x30)
    Label (312,676 206x40), "High temp. alarm diff (AHR)"
    Textfield (527,683 78x25), "%1.1f °C", tooltip "Provision_1.Low_temperature_alarm_differential", text variable: Provision_1.Low_temperature_alarm_differential
        p4168582468: Provision_1.Low_temperature_alarm_differential
    Rectangle (310,714 300x30)
    Label (312,709 208x40), "Probe temp alarm det. (ATI)"
    Textfield (527,716 78x25), "%1.0f Bar", tooltip "Provision_1.Probe_used_for_temperature_alarm_detection", text variable: Provision_1.Probe_used_for_temperature_alarm_detection
        p4168582468: Provision_1.Probe_used_for_temperature_alarm_detection
    Rectangle (310,293 300x30)
    Label (312,288 207x40), "Temp. alarm delay (ATD)"
    Textfield (527,295 78x25), "%1.2f min", tooltip "Provision_1.Temperature_alarm_delay", text variable: Provision_1.Temperature_alarm_delay
        p4168582468: Provision_1.Temperature_alarm_delay
        OnMouseClick: write the text variable via Default
    Rectangle (310,747 300x30)
    Label (312,742 205x40), "Op. high cond alarm (AHM)"
    Textfield (527,749 78x25), "%1.0f", tooltip "Provision_1.Operation_in_case_of_high_condenser_alarm", text variable: Provision_1.Operation_in_case_of_high_condenser_alarm
        p4168582468: Provision_1.Operation_in_case_of_high_condenser_alarm
    Rectangle (310,780 300x30)
    Label (313,775 205x40), "Cond. temp alarm (AHT)"
    Textfield (527,782 78x25), "%1.0f °C", tooltip "Provision_1.High_condenser_temperature", text variable: Provision_1.High_condenser_temperature
        p4168582468: Provision_1.High_condenser_temperature
    Rectangle (620,196 300x30)
    Label (621,191 209x40), "Door switch input mode (DSM)"
    Textfield (837,198 78x25), "%1.0f", tooltip "Provision_1.Door_switch_input_mode", text variable: Provision_1.Door_switch_input_mode
        p4168582468: Provision_1.Door_switch_input_mode
        OnMouseClick: write the text variable via Default
    Rectangle (932,326 300x30)
    Label (933,325 216x32), "RL4 output operation (OA4)"
    Textfield (1149,328 78x25), "%1.0f", tooltip "Provision_1.RL4_output_operation", text variable: Provision_1.RL4_output_operation
        p4168582468: Provision_1.RL4_output_operation
        OnMouseClick: write the text variable via Default
    Rectangle (310,227 300x30)
    Label (312,222 216x40), "Low temp alarm thresh. (ALA)"
    Textfield (527,229 78x25), "%1.0f °C", tooltip "Provision_1.Low_temperature_alarm_threshold", text variable: Provision_1.Low_temperature_alarm_threshold
        p4168582468: Provision_1.Low_temperature_alarm_threshold
        OnMouseClick: write the text variable via Default
    Rectangle (0,394 300x30)
    Label (1,389 211x40), "C/H output ON T1 faulty (CT1)"
    Textfield (217,396 78x25), "%1.0f min", tooltip "Provision_1.CH_output_ON_when_probe_T1_is_faulty", text variable: Provision_1.CH_output_ON_when_probe_T1_is_faulty
        p4168582468: Provision_1.CH_output_ON_when_probe_T1_is_faulty
        OnMouseClick: write the text variable via Default
    Rectangle (0,427 300x30)
    Label (1,423 210x40), "C/H output OFF T1 faulty (CT2)(CT2)"
    Textfield (217,429 78x25), "%1.0f min", tooltip "Provision_1.CH_output_OFF_when_probe_T1_is_faulty", text variable: Provision_1.CH_output_OFF_when_probe_T1_is_faulty
        p4168582468: Provision_1.CH_output_OFF_when_probe_T1_is_faulty
        OnMouseClick: write the text variable via Default
    Rectangle (311,460 300x30)
    Label (313,455 209x40), "Defrost interval (DFT)"
    Textfield (528,462 78x25), "%1.0f hour", tooltip "Provision_1.Time_based_defrost", text variable: Provision_1.Time_based_defrost
        p4168582468: Provision_1.Time_based_defrost
    Rectangle (1,460 300x30)
    Label (3,455 211x40), "Min time between defrost (DDS)"
    Textfield (218,462 78x25), "%1.2f hour", tooltip "Provision_1.Minimum_Time_Between_Defrost", text variable: Provision_1.Minimum_Time_Between_Defrost
        p4168582468: Provision_1.Minimum_Time_Between_Defrost
        OnMouseClick: write the text variable via Default
    Rectangle (310,326 300x30)
    Label (312,329 218x24), "Defrost type (DTY)"
    Textfield (527,328 78x25), "%1.0f", tooltip "Provision_1.Defrost_type", text variable: Provision_1.Defrost_type
        p4168582468: Provision_1.Defrost_type
        OnMouseClick: write the text variable via Default
    Rectangle (0,549 300x30)
    Label (2,544 210x40), "Delay for Hot Gas (DPD"
    Textfield (217,551 78x25), "%1.0f s", tooltip "Provision_1.Delay_for_pressure_equalization_for_hot_gas", text variable: Provision_1.Delay_for_pressure_equalization_for_hot_gas
        p4168582468: Provision_1.Delay_for_pressure_equalization_for_hot_gas
    Rectangle (310,359 300x30)
    Label (312,354 212x40), "Derfrost end temp (DLI)"
    Textfield (527,361 78x25), "%1.1f °C", tooltip "Provision_1.Defrost_end_temperature", text variable: Provision_1.Defrost_end_temperature
        p4168582468: Provision_1.Defrost_end_temperature
        OnMouseClick: write the text variable via Default
    Rectangle (310,392 300x30)
    Label (312,387 206x40), "Max defrost duration (DTO)"
    Textfield (527,394 78x25), "%1.0f min", tooltip "Provision_1.Maximum_defrost_duration", text variable: Provision_1.Maximum_defrost_duration
        p4168582468: Provision_1.Maximum_defrost_duration
        OnMouseClick: write the text variable via Default
    Rectangle (1,516 300x30)
    Label (2,511 210x40), "Defrost start mode (DFM)"
    Textfield (218,518 78x25), "%1.0f", tooltip "Provision_1.Defrost_start_mode", text variable: Provision_1.Defrost_start_mode
        p4168582468: Provision_1.Defrost_start_mode
    Rectangle (620,460 300x30)
    Label (622,462 211x26), "Defrost time optimiz. (DAR)"
    Textfield (837,462 78x25), "%1.0f", tooltip "Provision_1.Defrost_time_optimization", text variable: Provision_1.Defrost_time_optimization
        p4168582468: Provision_1.Defrost_time_optimization
        OnMouseClick: write the text variable via Default
    Rectangle (620,229 300x30)
    Label (621,224 210x40), "Door alarm delay (DAD)"
    Textfield (837,231 78x25), "%1.0f min", tooltip "Provision_1.Door_alarm_delay", text variable: Provision_1.Door_alarm_delay
        p4168582468: Provision_1.Door_alarm_delay
        OnMouseClick: write the text variable via Default
    Rectangle (621,683 300x30)
    Label (622,678 211x40), "Delay min / max temp logging"
    Textfield (838,685 78x25), "%1.0f sec", tooltip "Provision_1.Delay_for_minimum_and_maximum_temperature_logging", text variable: Provision_1.Delay_for_minimum_and_maximum_temperature_logging
        p4168582468: Provision_1.Delay_for_minimum_and_maximum_temperature_logging
    Rectangle (621,749 300x30)
    Label (623,744 210x40), "The rel. weight T2 / T1 (AVG)"
    Textfield (838,751 78x25), "%1.2f %%", tooltip "Provision_1.The_relative_weight_of_T2_on_T1", text variable: Provision_1.The_relative_weight_of_T2_on_T1
        p4168582468: Provision_1.The_relative_weight_of_T2_on_T1
    Rectangle (931,97 300x30)
    Label (933,92 210x40), "Display slow down (SIM)"
    Textfield (1148,99 78x25), "%1.0f", tooltip "Provision_1.Display_slowdown", text variable: Provision_1.Display_slowdown
        p4168582468: Provision_1.Display_slowdown
        OnMouseClick: write the text variable via Default
    Rectangle (931,130 300x30)
    Label (933,125 216x40), "Address PC com. (ADDR)"
    Textfield (1148,132 78x25), "%1.0f", tooltip "Provision_1.Address_for_PC_communication", text variable: Provision_1.Address_for_PC_communication
        p4168582468: Provision_1.Address_for_PC_communication
        OnMouseClick: write the text variable via Default
    Rectangle (621,716 300x30)
    Label (622,711 211x40), "Sel. temp. probe disp. (TDS)"
    Textfield (838,718 78x25), "%1.0f", tooltip "Provision_1.Selects_the_temperature_probe_to_be_displayed", text variable: Provision_1.Selects_the_temperature_probe_to_be_displayed
        p4168582468: Provision_1.Selects_the_temperature_probe_to_be_displayed
    Rectangle (931,162 300x30)
    Label (933,157 208x40), "Modbus protocol sel. (PRT)"
    Textfield (1148,164 78x25), "%1.0f", tooltip "Provision_1.Modbus_protocol_selection", text variable: Provision_1.Modbus_protocol_selection
        p4168582468: Provision_1.Modbus_protocol_selection
        OnMouseClick: write the text variable via Default
    Rectangle (1,583 300x30)
    Label (3,578 209x40), "Display defrost mode (DDM)"
    Textfield (218,585 78x25), "%1.0f", tooltip "Provision_1.Display_defrost_mode", text variable: Provision_1.Display_defrost_mode
        p4168582468: Provision_1.Display_defrost_mode
    Rectangle (621,98 300x30)
    Label (623,93 211x40), "Display slow down (DDY)"
    Textfield (838,100 78x25), "%1.2f min", tooltip "Provision_1.Display_delay", text variable: Provision_1.Display_delay
        p4168582468: Provision_1.Display_delay
        OnMouseClick: write the text variable via Default
    Rectangle (621,164 300x30)
    Label (623,167 218x24), "Fan restart temperature (FDD)"
    Textfield (838,166 78x25), "%1.1f °C", tooltip "Provision_1.Fan_restart_temperature_after_defrost", text variable: Provision_1.Fan_restart_temperature_after_defrost
        p4168582468: Provision_1.Fan_restart_temperature_after_defrost
        OnMouseClick: write the text variable via Default
    Rectangle (311,425 300x30)
    Label (312,420 210x40), "Drain down time (DRN)"
    Textfield (528,427 78x25), "%1.0f min", tooltip "Provision_1.Drain_down_time", text variable: Provision_1.Drain_down_time
        p4168582468: Provision_1.Drain_down_time
        OnMouseClick: write the text variable via Default
    Rectangle (621,131 300x30)
    Label (623,133 211x26), "Fans active during defr. (FID)"
    Textfield (838,133 78x25), "%1.0f", tooltip "Provision_1.Fans_active_during_defrost", text variable: Provision_1.Fans_active_during_defrost
        p4168582468: Provision_1.Fans_active_during_defrost
        OnMouseClick: write the text variable via Default
    Rectangle (1240,127 150x30)
    Rectangle (1240,160 150x30)
    Rectangle (1240,193 150x30)
    Rectangle (1240,226 150x30)
    Rectangle (1240,259 150x30)
    Rectangle (1240,292 150x30)
    Rectangle (1240,325 150x30)
    Lamp1 (1363,133 23x20), tooltip "Provision_1.dig1", variable: Provision_1.dig1, style: Lamp-Lamp1-Green
    Label (1240,129 112x26), "Digital in 1"
    Label (1240,165 105x21), "Digital in 2"
    Lamp1 (1363,166 23x20), tooltip "Provision_1.dig2", variable: Provision_1.dig2, style: Lamp-Lamp1-Green
    Label (1240,198 105x21), "Alarm"
    Lamp1 (1363,199 23x20), tooltip "Provision_1.alarm", variable: Provision_1.alarm, style: Lamp-Lamp1-Green
    Label (1240,231 105x21), "Alarm muted"
    Lamp1 (1363,232 23x20), tooltip "Provision_1.buzzer_mute", variable: Provision_1.buzzer_mute, style: Lamp-Lamp1-Green
    Label (1240,264 105x21), "Defrost"
    Lamp1 (1363,265 23x20), tooltip "Provision_1.defrost", variable: Provision_1.defrost, style: Lamp-Lamp1-Green
    Label (1240,297 130x21), "Door Open"
    Lamp1 (1363,298 23x20), tooltip "Provision_1.door_open", variable: Provision_1.door_open, style: Lamp-Lamp1-Green
    Lamp1 (1363,331 23x20), tooltip "Provision_1.test", variable: Provision_1.test, style: Lamp-Lamp1-Green
    Label (1240,330 111x21), "Test"
    Rectangle (1242,358 150x30)
    Rectangle (1396,129 150x30)
    Rectangle (1396,162 150x30)
    Rectangle (1396,195 150x30)
    Rectangle (1396,228 150x30)
    Rectangle (1396,261 150x30)
    Rectangle (1396,294 150x30)
    Lamp1 (1365,364 23x20), tooltip "Provision_1.machine_standby", variable: Provision_1.machine_standby, style: Lamp-Lamp1-Green
    Label (1242,360 112x26), "Standby"
    Label (1396,134 105x21), "T1 probe fail"
    Lamp1 (1519,135 23x20), tooltip "Provision_1.T1_failure", variable: Provision_1.T1_failure, style: Lamp-Lamp1-Red
    Label (1396,167 105x21), "T2 probe fail"
    Lamp1 (1519,168 23x20), tooltip "Provision_1.T2_failure", variable: Provision_1.T2_failure, style: Lamp-Lamp1-Red
    Label (1396,200 105x21), "T3 probe fail"
    Lamp1 (1519,201 23x20), tooltip "Provision_1.T3_failure", variable: Provision_1.T3_failure, style: Lamp-Lamp1-Red
    Label (1396,233 105x21), "Low temp"
    Lamp1 (1519,234 23x20), tooltip "Provision_1.Low_temperature", variable: Provision_1.Low_temperature, style: Lamp-Lamp1-Red
    Label (1396,266 130x21), "High temp"
    Lamp1 (1519,267 23x20), tooltip "Provision_1.High_temperature", variable: Provision_1.High_temperature, style: Lamp-Lamp1-Red
    Lamp1 (1519,300 23x20), tooltip "Provision_1.High_condenser_temperature", variable: Provision_1.High_condenser_temperature, style: Lamp-Lamp1-Red
    Label (1396,299 111x21), "High cond temp"
    Rectangle (1396,327 150x30)
    Rectangle (1396,360 150x30)
    Label (1396,332 105x21), "Generic"
    Lamp1 (1519,333 23x20), tooltip "Provision_1.Generic_alarm", variable: Provision_1.Generic_alarm, style: Lamp-Lamp1-Red
    Label (1396,365 105x21), "Door open"
    Lamp1 (1519,366 23x20), tooltip "Provision_1.Door_open_alarm", variable: Provision_1.Door_open_alarm, style: Lamp-Lamp1-Red
    Rectangle (1395,96 151x30)
    Label (1396,94 162x30), "Alarm"
    Rectangle (1240,94 151x30)
    Label (1241,94 162x30), "Status"
    Button (933,427 124x30), "Read Parameters"
        OnMouseClick:  ToggleVariable=Provision_1.read_param_button
        OnMouseDown:  ToggleVariable=Provision_1.xtrigger_get_param
        OnMouseUp:  ToggleVariable=Provision_1.xtrigger_get_param
        OnMouseUp:  ToggleVariable=Provision_1.all_param_read
    Label (930,514 294x30), "Non changeable parameters"
    Label (930,362 294x30), "Changeable parameters"
    Button (1073,427 124x30), "Set Parameters"
        OnMouseDown:  ToggleVariable=Provision_1.xtrigger_set_param
        OnMouseUp:  ToggleVariable=Provision_1.xtrigger_set_param
    Rectangle (932,387 300x30)
    Label (933,386 216x32), "parameter read delay"
    Textfield (1120,389 107x25), "%t[ss:ms]", tooltip "Provision_1.RL4_output_operation", text variable: Provision_1.set_delaytime
        p4168582468: Provision_1.set_delaytime
        OnMouseClick: write the text variable via Default
END_VISUALIZATION

// Device/Application/Provision_overview
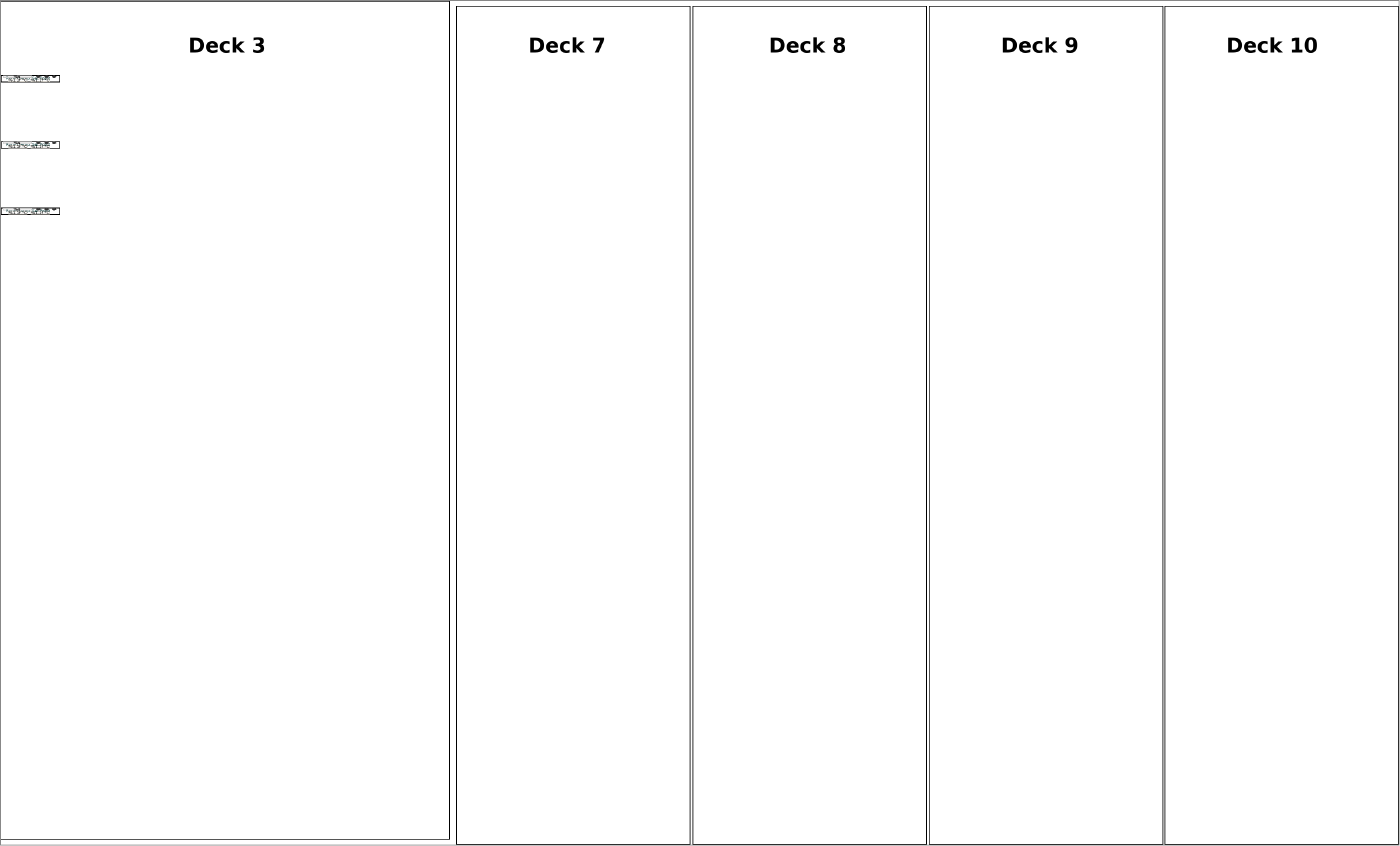
VISUALIZATION Provision_overview  // 1688x1021
    Rectangle (1404,7 282x1012)
    Rectangle (1120,7 282x1012)
    Rectangle (550,7 282x1012)
    Rectangle (835,7 282x1012)
    Rectangle (-5,1 547x1012)
    Label (199,40 150x30), "Deck 3"
    Label (609,40 150x30), "Deck 7"
    Label (899,40 150x30), "Deck 8"
    Label (1179,40 150x30), "Deck 9"
    Label (1459,40 150x30), "Deck 10"
    Frame (0,90 272x85)
        shows ProvRoomTemp(provroomTemp := Main_program.Provision_room1)
    Frame (0,250 272x85)
        shows ProvRoomTemp(provroomTemp := Main_program.Provision_room3)
    Frame (0,170 272x85)
        shows ProvRoomTemp(provroomTemp := Main_program.Provision_room2)
END_VISUALIZATION

